LIN {X 0,Y 298.192,Z 478.827,A -85,B 0,C 180,E1 -16627.38,E2 -16627.38} C_VEL
LIN {X 0,Y 298.477,Z 490.19,A -85,B 0,C 180,E1 -16628.776,E2 -16628.776} C_VEL
LIN {X 0,Y 297.905,Z 495.3,A -85,B 0,C 180,E1 -16629.456,E2 -16629.456} C_VEL
LIN {X 0,Y 296.112,Z 505.168,A -85,B 0,C 180,E1 -16630.953,E2 -16630.953} C_VEL
LIN {X 0,Y 294.392,Z 514.617,A -85,B 0,C 180,E1 -16632.731,E2 -16632.731} C_VEL
LIN {X 0,Y 292.913,Z 523.059,A -85,B 0,C 180,E1 -16634.697,E2 -16634.697} C_VEL
LIN {X 0,Y 291.619,Z 530.199,A -85,B 0,C 180,E1 -16636.765,E2 -16636.765} C_VEL
LIN {X 0,Y 290.674,Z 535.95,A -85,B 0,C 180,E1 -16638.847,E2 -16638.847} C_VEL
LIN {X 0,Y 290.055,Z 540.511,A -85,B 0,C 180,E1 -16640.938,E2 -16640.938} C_VEL
LIN {X 0,Y 289.711,Z 543.998,A -85,B 0,C 180,E1 -16643.033,E2 -16643.033} C_VEL
LIN {X 0,Y 289.605,Z 545.749,A -85,B 0,C 180,E1 -16644.429,E2 -16644.429} C_VEL
LIN {X 0,Y 289.581,Z 547.097,A -85,B 0,C 180,E1 -16645.824,E2 -16645.824} C_VEL
LIN {X 0,Y 289.556,Z 548.044,A -85,B 0,C 180,E1 -16647.217,E2 -16647.217} C_VEL
LIN {X 0,Y 289.58,Z 548.554,A -85,B 0,C 180,E1 -16648.609,E2 -16648.609} C_VEL
LIN {X 0,Y 289.708,Z 548.659,A -85,B 0,C 180,E1 -16650,E2 -16650} C_VEL
LIN {X 0,Y 289.61,Z 548.356,A -85,B 0,C 180,E1 -16651.39,E2 -16651.39} C_VEL
LIN {X 0,Y 289.566,Z 547.661,A -85,B 0,C 180,E1 -16652.782,E2 -16652.782} C_VEL
LIN {X 0,Y 289.603,Z 546.528,A -85,B 0,C 180,E1 -16654.175,E2 -16654.175} C_VEL
LIN {X 0,Y 289.638,Z 544.641,A -85,B 0,C 180,E1 -16655.813,E2 -16655.813} C_VEL
LIN {X 0,Y 289.906,Z 540.509,A -85,B 0,C 180,E1 -16658.363,E2 -16658.363} C_VEL
LIN {X 0,Y 290.445,Z 535.873,A -85,B 0,C 180,E1 -16660.455,E2 -16660.455} C_VEL
LIN {X 0,Y 291.359,Z 528.848,A -85,B 0,C 180,E1 -16662.892,E2 -16662.892} C_VEL
LIN {X 0,Y 292.574,Z 521.257,A -85,B 0,C 180,E1 -16664.964,E2 -16664.964} C_VEL
LIN {X 0,Y 294.049,Z 512.473,A -85,B 0,C 180,E1 -16666.878,E2 -16666.878} C_VEL
LIN {X 0,Y 295.452,Z 501.889,A -85,B 0,C 180,E1 -16668.73,E2 -16668.73} C_VEL
LIN {X 0,Y 297.226,Z 490.969,A -85,B 0,C 180,E1 -16670.231,E2 -16670.231} C_VEL
LIN {X 0,Y 296.981,Z 482.707,A -85,B 0,C 180,E1 -16671.232,E2 -16671.232} C_VEL
LIN {X 0,Y 296.01,Z 470.906,A -85,B 0,C 180,E1 -16672.452,E2 -16672.452} C_VEL
LIN {X 0,Y 294.301,Z 457.671,A -85,B 0,C 180,E1 -16673.542,E2 -16673.542} C_VEL
LIN {X 0,Y 291.805,Z 444.082,A -85,B 0,C 180,E1 -16674.412,E2 -16674.412} C_VEL
LIN {X 0,Y 291.28,Z 441.289,A -85,B 0,C 180,E1 -16674.556,E2 -16674.556} C_VEL
LIN {X 0,Y 291.996,Z 435.686,A -85,B 0,C 180,E1 -16677.991,E2 -16677.991} C_VEL
LIN {X 0,Y 292.755,Z 430.711,A -85,B 0,C 180,E1 -16681.072,E2 -16681.072} C_VEL
LIN {X 0,Y 293.852,Z 424.513,A -85,B 0,C 180,E1 -16685.029,E2 -16685.029} C_VEL
LIN {X 0,Y 294.193,Z 422.009,A -85,B 0,C 180,E1 -16686.67,E2 -16686.67} C_VEL
LIN {X 0,Y 293.916,Z 418.336,A -85,B 0,C 180,E1 -16689.213,E2 -16689.213} C_VEL
LIN {X 0,Y 293.01,Z 413.146,A -85,B 0,C 180,E1 -16693.054,E2 -16693.054} C_VEL
LIN {X 0,Y 292.263,Z 409.186,A -85,B 0,C 180,E1 -16696.169,E2 -16696.169} C_VEL
LIN {X 0,Y 291.395,Z 404.188,A -85,B 0,C 180,E1 -16700.418,E2 -16700.418} C_VEL
LIN {X 0,Y 291.423,Z 404.186,A -85,B 0,C 180,E1 -16702.922,E2 -16702.922} C_VEL
LIN {X 0,Y 291.339,Z 404.193,A -85,B 0,C 180,E1 -16706.301,E2 -16706.301} C_VEL
LIN {X 0,Y 291.378,Z 404.189,A -85,B 0,C 180,E1 -16710.261,E2 -16710.261} C_VEL
LIN {X 0,Y 291.406,Z 404.185,A -85,B 0,C 180,E1 -16714.271,E2 -16714.271} C_VEL
LIN {X 0,Y 291.375,Z 404.189,A -85,B 0,C 180,E1 -16717.299,E2 -16717.299} C_VEL
LIN {X 0,Y 291.452,Z 404.179,A -85,B 0,C 180,E1 -16720.27,E2 -16720.27} C_VEL
LIN {X 0,Y 291.549,Z 404.17,A -85,B 0,C 180,E1 -16724.623,E2 -16724.623} C_VEL
LIN {X 0,Y 291.528,Z 404.172,A -85,B 0,C 180,E1 -16728.88,E2 -16728.88} C_VEL
LIN {X 0,Y 291.68,Z 404.149,A -85,B 0,C 180,E1 -16731.688,E2 -16731.688} C_VEL
LIN {X 0,Y 291.62,Z 404.158,A -85,B 0,C 180,E1 -16734.468,E2 -16734.468} C_VEL
LIN {X 0,Y 291.884,Z 404.129,A -85,B 0,C 180,E1 -16738.62,E2 -16738.62} C_VEL
LIN {X 0,Y 291.884,Z 404.123,A -85,B 0,C 180,E1 -16741.38,E2 -16741.38} C_VEL
LIN {X 0,Y 291.739,Z 404.144,A -85,B 0,C 180,E1 -16746.918,E2 -16746.918} C_VEL
LIN {X 0,Y 291.623,Z 404.156,A -85,B 0,C 180,E1 -16749.712,E2 -16749.712} C_VEL
LIN {X 0,Y 291.515,Z 404.167,A -85,B 0,C 180,E1 -16753.951,E2 -16753.951} C_VEL
LIN {X 0,Y 291.48,Z 404.176,A -85,B 0,C 180,E1 -16756.818,E2 -16756.818} C_VEL
LIN {X 0,Y 291.445,Z 404.179,A -85,B 0,C 180,E1 -16759.876,E2 -16759.876} C_VEL
LIN {X 0,Y 291.395,Z 404.185,A -85,B 0,C 180,E1 -16764.206,E2 -16764.206} C_VEL
LIN {X 0,Y 291.417,Z 404.182,A -85,B 0,C 180,E1 -16767.272,E2 -16767.272} C_VEL
LIN {X 0,Y 291.332,Z 404.194,A -85,B 0,C 180,E1 -16770.438,E2 -16770.438} C_VEL
LIN {X 0,Y 291.34,Z 404.19,A -85,B 0,C 180,E1 -16773.699,E2 -16773.699} C_VEL
LIN {X 0,Y 291.397,Z 404.185,A -85,B 0,C 180,E1 -16777.261,E2 -16777.261} C_VEL
LIN {X 0,Y 291.373,Z 404.186,A -85,B 0,C 180,E1 -16780.636,E2 -16780.636} C_VEL
LIN {X 0,Y 291.296,Z 404.201,A -85,B 0,C 180,E1 -16784.401,E2 -16784.401} C_VEL
LIN {X 0,Y 291.324,Z 404.194,A -85,B 0,C 180,E1 -16788.405,E2 -16788.405} C_VEL
LIN {X 0,Y 291.346,Z 404.184,A -85,B 0,C 180,E1 -16791.159,E2 -16791.159} C_VEL
LIN {X 0,Y 291.36,Z 404.188,A -85,B 0,C 180,E1 -16794.627,E2 -16794.627} C_VEL
LIN {X 0,Y 291.371,Z 404.193,A -85,B 0,C 180,E1 -16797.952,E2 -16797.952} C_VEL
LIN {X 0,Y 291.377,Z 404.187,A -85,B 0,C 180,E1 -16801.159,E2 -16801.159} C_VEL
LIN {X 0,Y 291.417,Z 404.18,A -85,B 0,C 180,E1 -16804.273,E2 -16804.273} C_VEL
LIN {X 0,Y 291.383,Z 404.186,A -85,B 0,C 180,E1 -16807.301,E2 -16807.301} C_VEL
LIN {X 0,Y 291.46,Z 404.178,A -85,B 0,C 180,E1 -16810.271,E2 -16810.271} C_VEL
LIN {X 0,Y 291.557,Z 404.165,A -85,B 0,C 180,E1 -16814.624,E2 -16814.624} C_VEL
LIN {X 0,Y 291.54,Z 404.165,A -85,B 0,C 180,E1 -16818.881,E2 -16818.881} C_VEL
LIN {X 0,Y 291.713,Z 404.15,A -85,B 0,C 180,E1 -16821.689,E2 -16821.689} C_VEL
LIN {X 0,Y 291.617,Z 404.157,A -85,B 0,C 180,E1 -16824.469,E2 -16824.469} C_VEL
LIN {X 0,Y 291.827,Z 404.132,A -85,B 0,C 180,E1 -16828.62,E2 -16828.62} C_VEL
LIN {X 0,Y 290.81,Z 404.574,A -85,B 0,C 180,E1 -16831.385,E2 -16831.385} C_VEL
LIN {X 0,Y 290.925,Z 406.775,A -85,B 0,C 180,E1 -16834.156,E2 -16834.156} C_VEL
LIN {X 0,Y 290.743,Z 409.661,A -85,B 0,C 180,E1 -16837.718,E2 -16837.718} C_VEL
LIN {X 0,Y 294.779,Z 423.834,A -85,B 0,C 180,E1 -16838.772,E2 -16838.772} C_VEL
LIN {X 0,Y 297.668,Z 435.363,A -85,B 0,C 180,E1 -16839.841,E2 -16839.841} C_VEL
LIN {X 0,Y 299.398,Z 444.412,A -85,B 0,C 180,E1 -16840.824,E2 -16840.824} C_VEL
LIN {X 0,Y 298.317,Z 455.723,A -85,B 0,C 180,E1 -16842.069,E2 -16842.069} C_VEL
LIN {X 0,Y 296.897,Z 466.255,A -85,B 0,C 180,E1 -16843.518,E2 -16843.518} C_VEL
LIN {X 0,Y 295.437,Z 475.921,A -85,B 0,C 180,E1 -16845.169,E2 -16845.169} C_VEL
LIN {X 0,Y 293.98,Z 484.669,A -85,B 0,C 180,E1 -16847.008,E2 -16847.008} C_VEL
LIN {X 0,Y 292.804,Z 491.976,A -85,B 0,C 180,E1 -16848.907,E2 -16848.907} C_VEL
LIN {X 0,Y 291.692,Z 498.923,A -85,B 0,C 180,E1 -16851.187,E2 -16851.187} C_VEL
LIN {X 0,Y 290.88,Z 504.062,A -85,B 0,C 180,E1 -16853.346,E2 -16853.346} C_VEL
LIN {X 0,Y 290.305,Z 508.488,A -85,B 0,C 180,E1 -16855.834,E2 -16855.834} C_VEL
LIN {X 0,Y 289.944,Z 510.535,A -85,B 0,C 180,E1 -16857.422,E2 -16857.422} C_VEL
LIN {X 0,Y 289.668,Z 512.157,A -85,B 0,C 180,E1 -16859.138,E2 -16859.138} C_VEL
LIN {X 0,Y 289.52,Z 513.41,A -85,B 0,C 180,E1 -16861.83,E2 -16861.83} C_VEL
LIN {X 0,Y 289.676,Z 513.225,A -85,B 0,C 180,E1 -16864.422,E2 -16864.422} C_VEL
LIN {X 0,Y 290.085,Z 511.76,A -85,B 0,C 180,E1 -16866.917,E2 -16866.917} C_VEL
LIN {X 0,Y 290.713,Z 509.081,A -85,B 0,C 180,E1 -16869.321,E2 -16869.321} C_VEL
LIN {X 0,Y 291.454,Z 505.271,A -85,B 0,C 180,E1 -16871.623,E2 -16871.623} C_VEL
LIN {X 0,Y 292.66,Z 499.549,A -85,B 0,C 180,E1 -16874.139,E2 -16874.139} C_VEL
LIN {X 0,Y 294.138,Z 492.812,A -85,B 0,C 180,E1 -16876.383,E2 -16876.383} C_VEL
LIN {X 0,Y 295.697,Z 485.104,A -85,B 0,C 180,E1 -16878.402,E2 -16878.402} C_VEL
LIN {X 0,Y 297.506,Z 475.704,A -85,B 0,C 180,E1 -16880.37,E2 -16880.37} C_VEL
LIN {X 0,Y 299.342,Z 465.228,A -85,B 0,C 180,E1 -16882.099,E2 -16882.099} C_VEL
LIN {X 0,Y 300.836,Z 455.272,A -85,B 0,C 180,E1 -16883.422,E2 -16883.422} C_VEL
LIN {X 0,Y 301.696,Z 448.206,A -85,B 0,C 180,E1 -16884.216,E2 -16884.216} C_VEL
LIN {X 0,Y 299.573,Z 437.974,A -85,B 0,C 180,E1 -16885.479,E2 -16885.479} C_VEL
LIN {X 0,Y 296.301,Z 426.472,A -85,B 0,C 180,E1 -16886.735,E2 -16886.735} C_VEL
LIN {X 0,Y 291.875,Z 414.797,A -85,B 0,C 180,E1 -16887.902,E2 -16887.902} C_VEL
LIN {X 0,Y 290.942,Z 412.026,A -85,B 0,C 180,E1 -16888.152,E2 -16888.152} C_VEL
LIN {X 0,Y 291.119,Z 409.938,A -85,B 0,C 180,E1 -16891.13,E2 -16891.13} C_VEL
LIN {X 0,Y 291.343,Z 407.807,A -85,B 0,C 180,E1 -16894.265,E2 -16894.265} C_VEL
LIN {X 0,Y 291.463,Z 405.839,A -85,B 0,C 180,E1 -16897.306,E2 -16897.306} C_VEL
LIN {X 0,Y 291.455,Z 404.184,A -85,B 0,C 180,E1 -16900.27,E2 -16900.27} C_VEL
LIN {X 0,Y 291.538,Z 404.173,A -85,B 0,C 180,E1 -16904.634,E2 -16904.634} C_VEL
LIN {X 0,Y 291.532,Z 404.17,A -85,B 0,C 180,E1 -16908.88,E2 -16908.88} C_VEL
LIN {X 0,Y 291.682,Z 404.153,A -85,B 0,C 180,E1 -16911.815,E2 -16911.815} C_VEL
LIN {X 0,Y 291.623,Z 404.157,A -85,B 0,C 180,E1 -16914.468,E2 -16914.468} C_VEL
LIN {X 0,Y 291.806,Z 404.133,A -85,B 0,C 180,E1 -16917.797,E2 -16917.797} C_VEL
LIN {X 0,Y 291.193,Z 404.214,A -85,B 0,C 180,E1 -16918.951,E2 -16918.951} C_VEL
LIN {X 0,Y 288.337,Z 404.57,A -85,B 0,C 180,E1 -16920.827,E2 -16920.827} C_VEL
LIN {X 0,Y 285.826,Z 404.878,A -85,B 0,C 180,E1 -16922.35,E2 -16922.35} C_VEL
LIN {X 0,Y 284.673,Z 405.026,A -85,B 0,C 180,E1 -16923.531,E2 -16923.531} C_VEL
LIN {X 0,Y 284.541,Z 405.039,A -85,B 0,C 180,E1 -16923.932,E2 -16923.932} C_VEL
LIN {X 0,Y 284.683,Z 405.023,A -85,B 0,C 180,E1 -16927.09,E2 -16927.09} C_VEL
LIN {X 0,Y 284.516,Z 405.043,A -85,B 0,C 180,E1 -16929.957,E2 -16929.957} C_VEL
LIN {X 0,Y 284.474,Z 405.049,A -85,B 0,C 180,E1 -16934.303,E2 -16934.303} C_VEL
LIN {X 0,Y 284.422,Z 405.056,A -85,B 0,C 180,E1 -16937.248,E2 -16937.248} C_VEL
LIN {X 0,Y 284.376,Z 405.063,A -85,B 0,C 180,E1 -16940.242,E2 -16940.242} C_VEL
LIN {X 0,Y 284.366,Z 405.065,A -85,B 0,C 180,E1 -16943.875,E2 -16943.875} C_VEL
LIN {X 0,Y 284.391,Z 405.059,A -85,B 0,C 180,E1 -16947.173,E2 -16947.173} C_VEL
LIN {X 0,Y 284.291,Z 405.073,A -85,B 0,C 180,E1 -16951.275,E2 -16951.275} C_VEL
LIN {X 0,Y 284.328,Z 405.111,A -85,B 0,C 180,E1 -16954.647,E2 -16954.647} C_VEL
LIN {X 0,Y 284.864,Z 407.869,A -85,B 0,C 180,E1 -16958.082,E2 -16958.082} C_VEL
LIN {X 0,Y 285.385,Z 411.197,A -85,B 0,C 180,E1 -16961.676,E2 -16961.676} C_VEL
LIN {X 0,Y 286.093,Z 415.045,A -85,B 0,C 180,E1 -16965.43,E2 -16965.43} C_VEL
LIN {X 0,Y 286.915,Z 419.566,A -85,B 0,C 180,E1 -16969.407,E2 -16969.407} C_VEL
LIN {X 0,Y 287.353,Z 423.183,A -85,B 0,C 180,E1 -16972.307,E2 -16972.307} C_VEL
LIN {X 0,Y 286.992,Z 426.701,A -85,B 0,C 180,E1 -16974.867,E2 -16974.867} C_VEL
LIN {X 0,Y 285.711,Z 433.39,A -85,B 0,C 180,E1 -16979.422,E2 -16979.422} C_VEL
LIN {X 0,Y 284.749,Z 439.073,A -85,B 0,C 180,E1 -16983.131,E2 -16983.131} C_VEL
LIN {X 0,Y 288.298,Z 453.543,A -85,B 0,C 180,E1 -16984.266,E2 -16984.266} C_VEL
LIN {X 0,Y 290.471,Z 465.856,A -85,B 0,C 180,E1 -16985.414,E2 -16985.414} C_VEL
LIN {X 0,Y 291.465,Z 477.28,A -85,B 0,C 180,E1 -16986.627,E2 -16986.627} C_VEL
LIN {X 0,Y 291.721,Z 488.901,A -85,B 0,C 180,E1 -16988.074,E2 -16988.074} C_VEL
LIN {X 0,Y 291.496,Z 494.105,A -85,B 0,C 180,E1 -16988.798,E2 -16988.798} C_VEL
LIN {X 0,Y 289.389,Z 505.1,A -85,B 0,C 180,E1 -16990.493,E2 -16990.493} C_VEL
LIN {X 0,Y 287.468,Z 515.166,A -85,B 0,C 180,E1 -16992.453,E2 -16992.453} C_VEL
LIN {X 0,Y 286.029,Z 522.874,A -85,B 0,C 180,E1 -16994.319,E2 -16994.319} C_VEL
LIN {X 0,Y 284.693,Z 529.951,A -85,B 0,C 180,E1 -16996.437,E2 -16996.437} C_VEL
LIN {X 0,Y 283.675,Z 535.656,A -85,B 0,C 180,E1 -16998.568,E2 -16998.568} C_VEL
LIN {X 0,Y 282.999,Z 540.176,A -85,B 0,C 180,E1 -17000.71,E2 -17000.71} C_VEL
LIN {X 0,Y 282.63,Z 543.631,A -85,B 0,C 180,E1 -17002.858,E2 -17002.858} C_VEL
LIN {X 0,Y 282.543,Z 545.371,A -85,B 0,C 180,E1 -17004.29,E2 -17004.29} C_VEL
LIN {X 0,Y 282.5,Z 546.707,A -85,B 0,C 180,E1 -17005.72,E2 -17005.72} C_VEL
LIN {X 0,Y 282.483,Z 547.638,A -85,B 0,C 180,E1 -17007.148,E2 -17007.148} C_VEL
LIN {X 0,Y 282.619,Z 548.22,A -85,B 0,C 180,E1 -17010,E2 -17010} C_VEL
LIN {X 0,Y 282.522,Z 547.905,A -85,B 0,C 180,E1 -17011.425,E2 -17011.425} C_VEL
LIN {X 0,Y 282.493,Z 547.195,A -85,B 0,C 180,E1 -17012.852,E2 -17012.852} C_VEL
LIN {X 0,Y 282.521,Z 546.036,A -85,B 0,C 180,E1 -17014.279,E2 -17014.279} C_VEL
LIN {X 0,Y 282.558,Z 544.359,A -85,B 0,C 180,E1 -17015.782,E2 -17015.782} C_VEL
LIN {X 0,Y 282.739,Z 541.243,A -85,B 0,C 180,E1 -17017.857,E2 -17017.857} C_VEL
LIN {X 0,Y 283.214,Z 536.959,A -85,B 0,C 180,E1 -17020.003,E2 -17020.003} C_VEL
LIN {X 0,Y 284.043,Z 530.454,A -85,B 0,C 180,E1 -17022.503,E2 -17022.503} C_VEL
LIN {X 0,Y 285.283,Z 523.33,A -85,B 0,C 180,E1 -17024.625,E2 -17024.625} C_VEL
LIN {X 0,Y 286.742,Z 514.44,A -85,B 0,C 180,E1 -17026.737,E2 -17026.737} C_VEL
LIN {X 0,Y 288.055,Z 505.319,A -85,B 0,C 180,E1 -17028.491,E2 -17028.491} C_VEL
LIN {X 0,Y 289.673,Z 495.289,A -85,B 0,C 180,E1 -17030.041,E2 -17030.041} C_VEL
LIN {X 0,Y 290.456,Z 490.049,A -85,B 0,C 180,E1 -17030.724,E2 -17030.724} C_VEL
LIN {X 0,Y 289.724,Z 477.737,A -85,B 0,C 180,E1 -17032.208,E2 -17032.208} C_VEL
LIN {X 0,Y 288.577,Z 465.951,A -85,B 0,C 180,E1 -17033.36,E2 -17033.36} C_VEL
LIN {X 0,Y 286.64,Z 453.247,A -85,B 0,C 180,E1 -17034.36,E2 -17034.36} C_VEL
LIN {X 0,Y 284.317,Z 440.877,A -85,B 0,C 180,E1 -17035.141,E2 -17035.141} C_VEL
LIN {X 0,Y 285.104,Z 435.166,A -85,B 0,C 180,E1 -17038.729,E2 -17038.729} C_VEL
LIN {X 0,Y 285.884,Z 430.222,A -85,B 0,C 180,E1 -17041.906,E2 -17041.906} C_VEL
LIN {X 0,Y 286.829,Z 425.249,A -85,B 0,C 180,E1 -17045.155,E2 -17045.155} C_VEL
LIN {X 0,Y 287.146,Z 421.493,A -85,B 0,C 180,E1 -17047.724,E2 -17047.724} C_VEL
LIN {X 0,Y 286.6,Z 417.651,A -85,B 0,C 180,E1 -17050.52,E2 -17050.52} C_VEL
LIN {X 0,Y 285.695,Z 412.534,A -85,B 0,C 180,E1 -17054.488,E2 -17054.488} C_VEL
LIN {X 0,Y 284.666,Z 406.967,A -85,B 0,C 180,E1 -17059.138,E2 -17059.138} C_VEL
LIN {X 0,Y 284.34,Z 405.068,A -85,B 0,C 180,E1 -17060.929,E2 -17060.929} C_VEL
LIN {X 0,Y 284.357,Z 405.066,A -85,B 0,C 180,E1 -17064.645,E2 -17064.645} C_VEL
LIN {X 0,Y 284.288,Z 405.075,A -85,B 0,C 180,E1 -17068.725,E2 -17068.725} C_VEL
LIN {X 0,Y 284.388,Z 405.064,A -85,B 0,C 180,E1 -17072.827,E2 -17072.827} C_VEL
LIN {X 0,Y 284.36,Z 405.065,A -85,B 0,C 180,E1 -17076.706,E2 -17076.706} C_VEL
LIN {X 0,Y 284.397,Z 405.058,A -85,B 0,C 180,E1 -17081.261,E2 -17081.261} C_VEL
LIN {X 0,Y 284.486,Z 405.048,A -85,B 0,C 180,E1 -17084.459,E2 -17084.459} C_VEL
LIN {X 0,Y 284.48,Z 405.05,A -85,B 0,C 180,E1 -17088.601,E2 -17088.601} C_VEL
LIN {X 0,Y 284.632,Z 405.027,A -85,B 0,C 180,E1 -17091.48,E2 -17091.48} C_VEL
LIN {X 0,Y 284.591,Z 405.032,A -85,B 0,C 180,E1 -17094.331,E2 -17094.331} C_VEL
LIN {X 0,Y 284.85,Z 405.005,A -85,B 0,C 180,E1 -17098.586,E2 -17098.586} C_VEL
LIN {X 0,Y 284.85,Z 404.998,A -85,B 0,C 180,E1 -17101.414,E2 -17101.414} C_VEL
LIN {X 0,Y 284.691,Z 405.021,A -85,B 0,C 180,E1 -17107.09,E2 -17107.09} C_VEL
LIN {X 0,Y 284.56,Z 405.037,A -85,B 0,C 180,E1 -17109.956,E2 -17109.956} C_VEL
LIN {X 0,Y 284.471,Z 405.047,A -85,B 0,C 180,E1 -17114.304,E2 -17114.304} C_VEL
LIN {X 0,Y 284.419,Z 405.054,A -85,B 0,C 180,E1 -17117.249,E2 -17117.249} C_VEL
LIN {X 0,Y 284.373,Z 405.063,A -85,B 0,C 180,E1 -17120.243,E2 -17120.243} C_VEL
LIN {X 0,Y 284.363,Z 405.058,A -85,B 0,C 180,E1 -17123.876,E2 -17123.876} C_VEL
LIN {X 0,Y 284.392,Z 405.057,A -85,B 0,C 180,E1 -17127.174,E2 -17127.174} C_VEL
LIN {X 0,Y 284.291,Z 405.067,A -85,B 0,C 180,E1 -17131.275,E2 -17131.275} C_VEL
LIN {X 0,Y 284.358,Z 405.061,A -85,B 0,C 180,E1 -17135.355,E2 -17135.355} C_VEL
LIN {X 0,Y 284.329,Z 405.07,A -85,B 0,C 180,E1 -17138.167,E2 -17138.167} C_VEL
LIN {X 0,Y 284.289,Z 405.069,A -85,B 0,C 180,E1 -17141.873,E2 -17141.873} C_VEL
LIN {X 0,Y 284.253,Z 405.079,A -85,B 0,C 180,E1 -17146.19,E2 -17146.19} C_VEL
LIN {X 0,Y 284.304,Z 405.066,A -85,B 0,C 180,E1 -17150.025,E2 -17150.025} C_VEL
LIN {X 0,Y 284.329,Z 405.058,A -85,B 0,C 180,E1 -17153.615,E2 -17153.615} C_VEL
LIN {X 0,Y 284.307,Z 405.068,A -85,B 0,C 180,E1 -17157.191,E2 -17157.191} C_VEL
LIN {X 0,Y 284.355,Z 405.064,A -85,B 0,C 180,E1 -17160.377,E2 -17160.377} C_VEL
LIN {X 0,Y 284.378,Z 405.057,A -85,B 0,C 180,E1 -17163.588,E2 -17163.588} C_VEL
LIN {X 0,Y 284.368,Z 405.059,A -85,B 0,C 180,E1 -17166.708,E2 -17166.708} C_VEL
LIN {X 0,Y 284.405,Z 405.055,A -85,B 0,C 180,E1 -17171.263,E2 -17171.263} C_VEL
LIN {X 0,Y 284.494,Z 405.045,A -85,B 0,C 180,E1 -17174.46,E2 -17174.46} C_VEL
LIN {X 0,Y 284.491,Z 405.043,A -85,B 0,C 180,E1 -17178.602,E2 -17178.602} C_VEL
LIN {X 0,Y 284.663,Z 405.027,A -85,B 0,C 180,E1 -17181.482,E2 -17181.482} C_VEL
LIN {X 0,Y 284.59,Z 405.033,A -85,B 0,C 180,E1 -17184.332,E2 -17184.332} C_VEL
LIN {X 0,Y 284.789,Z 405.008,A -85,B 0,C 180,E1 -17188.586,E2 -17188.586} C_VEL
LIN {X 0,Y 283.768,Z 405.542,A -85,B 0,C 180,E1 -17191.42,E2 -17191.42} C_VEL
LIN {X 0,Y 283.887,Z 407.745,A -85,B 0,C 180,E1 -17194.259,E2 -17194.259} C_VEL
LIN {X 0,Y 283.716,Z 410.111,A -85,B 0,C 180,E1 -17197.161,E2 -17197.161} C_VEL
LIN {X 0,Y 287.713,Z 423.844,A -85,B 0,C 180,E1 -17198.217,E2 -17198.217} C_VEL
LIN {X 0,Y 290.911,Z 436.611,A -85,B 0,C 180,E1 -17199.439,E2 -17199.439} C_VEL
LIN {X 0,Y 292.666,Z 446.475,A -85,B 0,C 180,E1 -17200.551,E2 -17200.551} C_VEL
LIN {X 0,Y 291.37,Z 457.536,A -85,B 0,C 180,E1 -17201.831,E2 -17201.831} C_VEL
LIN {X 0,Y 289.792,Z 468.719,A -85,B 0,C 180,E1 -17203.462,E2 -17203.462} C_VEL
LIN {X 0,Y 288.273,Z 478.258,A -85,B 0,C 180,E1 -17205.194,E2 -17205.194} C_VEL
LIN {X 0,Y 286.801,Z 486.78,A -85,B 0,C 180,E1 -17207.119,E2 -17207.119} C_VEL
LIN {X 0,Y 285.431,Z 494.876,A -85,B 0,C 180,E1 -17209.415,E2 -17209.415} C_VEL
LIN {X 0,Y 284.35,Z 501.337,A -85,B 0,C 180,E1 -17211.761,E2 -17211.761} C_VEL
LIN {X 0,Y 283.56,Z 506.404,A -85,B 0,C 180,E1 -17214.191,E2 -17214.191} C_VEL
LIN {X 0,Y 283.032,Z 510.101,A -85,B 0,C 180,E1 -17216.629,E2 -17216.629} C_VEL
LIN {X 0,Y 282.706,Z 511.814,A -85,B 0,C 180,E1 -17218.186,E2 -17218.186} C_VEL
LIN {X 0,Y 282.518,Z 513.04,A -85,B 0,C 180,E1 -17219.836,E2 -17219.836} C_VEL
LIN {X 0,Y 282.432,Z 513.897,A -85,B 0,C 180,E1 -17222.214,E2 -17222.214} C_VEL
LIN {X 0,Y 282.656,Z 513.566,A -85,B 0,C 180,E1 -17224.881,E2 -17224.881} C_VEL
LIN {X 0,Y 283.124,Z 511.934,A -85,B 0,C 180,E1 -17227.407,E2 -17227.407} C_VEL
LIN {X 0,Y 283.882,Z 508.804,A -85,B 0,C 180,E1 -17230.066,E2 -17230.066} C_VEL
LIN {X 0,Y 284.618,Z 505.178,A -85,B 0,C 180,E1 -17232.201,E2 -17232.201} C_VEL
LIN {X 0,Y 285.781,Z 499.981,A -85,B 0,C 180,E1 -17234.506,E2 -17234.506} C_VEL
LIN {X 0,Y 287.313,Z 493.347,A -85,B 0,C 180,E1 -17236.771,E2 -17236.771} C_VEL
LIN {X 0,Y 289.111,Z 485.063,A -85,B 0,C 180,E1 -17238.978,E2 -17238.978} C_VEL
LIN {X 0,Y 291.009,Z 475.574,A -85,B 0,C 180,E1 -17240.987,E2 -17240.987} C_VEL
LIN {X 0,Y 292.814,Z 465.777,A -85,B 0,C 180,E1 -17242.626,E2 -17242.626} C_VEL
LIN {X 0,Y 294.471,Z 455.215,A -85,B 0,C 180,E1 -17244.051,E2 -17244.051} C_VEL
LIN {X 0,Y 295.117,Z 449.319,A -85,B 0,C 180,E1 -17244.737,E2 -17244.737} C_VEL
LIN {X 0,Y 292.891,Z 438.87,A -85,B 0,C 180,E1 -17246.09,E2 -17246.09} C_VEL
LIN {X 0,Y 289.435,Z 426.934,A -85,B 0,C 180,E1 -17247.466,E2 -17247.466} C_VEL
LIN {X 0,Y 285.051,Z 415.59,A -85,B 0,C 180,E1 -17248.663,E2 -17248.663} C_VEL
LIN {X 0,Y 283.974,Z 412.528,A -85,B 0,C 180,E1 -17248.959,E2 -17248.959} C_VEL
LIN {X 0,Y 284.248,Z 409.868,A -85,B 0,C 180,E1 -17252.884,E2 -17252.884} C_VEL
LIN {X 0,Y 284.444,Z 407.426,A -85,B 0,C 180,E1 -17256.713,E2 -17256.713} C_VEL
LIN {X 0,Y 284.435,Z 405.546,A -85,B 0,C 180,E1 -17259.87,E2 -17259.87} C_VEL
LIN {X 0,Y 284.395,Z 405.062,A -85,B 0,C 180,E1 -17261.261,E2 -17261.261} C_VEL
LIN {X 0,Y 284.475,Z 405.052,A -85,B 0,C 180,E1 -17264.469,E2 -17264.469} C_VEL
LIN {X 0,Y 284.484,Z 405.048,A -85,B 0,C 180,E1 -17268.601,E2 -17268.601} C_VEL
LIN {X 0,Y 284.636,Z 405.031,A -85,B 0,C 180,E1 -17271.48,E2 -17271.48} C_VEL
LIN {X 0,Y 284.594,Z 405.033,A -85,B 0,C 180,E1 -17274.331,E2 -17274.331} C_VEL
LIN {X 0,Y 284.852,Z 405.004,A -85,B 0,C 180,E1 -17278.586,E2 -17278.586} C_VEL
LIN {X 0,Y 284.853,Z 405.003,A -85,B 0,C 180,E1 -17281.414,E2 -17281.414} C_VEL
LIN {X 0,Y 284.541,Z 405.039,A -85,B 0,C 180,E1 -17283.932,E2 -17283.932} C_VEL
LIN {X 0,Y 283.79,Z 405.139,A -85,B 0,C 180,E1 -17285.114,E2 -17285.114} C_VEL
LIN {X 0,Y 280.97,Z 405.494,A -85,B 0,C 180,E1 -17287.041,E2 -17287.041} C_VEL
LIN {X 0,Y 278.61,Z 405.784,A -85,B 0,C 180,E1 -17288.606,E2 -17288.606} C_VEL
LIN {X 0,Y 277.564,Z 405.909,A -85,B 0,C 180,E1 -17289.816,E2 -17289.816} C_VEL
LIN {X 0,Y 277.457,Z 405.92,A -85,B 0,C 180,E1 -17290.226,E2 -17290.226} C_VEL
LIN {X 0,Y 277.425,Z 405.928,A -85,B 0,C 180,E1 -17294.675,E2 -17294.675} C_VEL
LIN {X 0,Y 277.342,Z 405.934,A -85,B 0,C 180,E1 -17299.234,E2 -17299.234} C_VEL
LIN {X 0,Y 277.316,Z 405.943,A -85,B 0,C 180,E1 -17304.17,E2 -17304.17} C_VEL
LIN {X 0,Y 277.32,Z 405.942,A -85,B 0,C 180,E1 -17307.504,E2 -17307.504} C_VEL
LIN {X 0,Y 277.27,Z 405.948,A -85,B 0,C 180,E1 -17310.482,E2 -17310.482} C_VEL
LIN {X 0,Y 277.261,Z 405.952,A -85,B 0,C 180,E1 -17313.496,E2 -17313.496} C_VEL
LIN {X 0,Y 277.826,Z 408.899,A -85,B 0,C 180,E1 -17317.381,E2 -17317.381} C_VEL
LIN {X 0,Y 278.331,Z 412.111,A -85,B 0,C 180,E1 -17321.035,E2 -17321.035} C_VEL
LIN {X 0,Y 279.094,Z 416.179,A -85,B 0,C 180,E1 -17325.165,E2 -17325.165} C_VEL
LIN {X 0,Y 279.918,Z 420.681,A -85,B 0,C 180,E1 -17329.248,E2 -17329.248} C_VEL
LIN {X 0,Y 280.368,Z 424.167,A -85,B 0,C 180,E1 -17332.111,E2 -17332.111} C_VEL
LIN {X 0,Y 280.333,Z 425.75,A -85,B 0,C 180,E1 -17333.345,E2 -17333.345} C_VEL
LIN {X 0,Y 279.461,Z 430.007,A -85,B 0,C 180,E1 -17336.409,E2 -17336.409} C_VEL
LIN {X 0,Y 278.326,Z 435.931,A -85,B 0,C 180,E1 -17340.502,E2 -17340.502} C_VEL
LIN {X 0,Y 277.875,Z 438.585,A -85,B 0,C 180,E1 -17342.279,E2 -17342.279} C_VEL
LIN {X 0,Y 279.538,Z 444.902,A -85,B 0,C 180,E1 -17342.776,E2 -17342.776} C_VEL
LIN {X 0,Y 282.351,Z 456.878,A -85,B 0,C 180,E1 -17343.849,E2 -17343.849} C_VEL
LIN {X 0,Y 284.115,Z 468.137,A -85,B 0,C 180,E1 -17344.977,E2 -17344.977} C_VEL
LIN {X 0,Y 284.962,Z 480.077,A -85,B 0,C 180,E1 -17346.342,E2 -17346.342} C_VEL
LIN {X 0,Y 285.022,Z 491.674,A -85,B 0,C 180,E1 -17347.912,E2 -17347.912} C_VEL
LIN {X 0,Y 284.429,Z 496.544,A -85,B 0,C 180,E1 -17348.626,E2 -17348.626} C_VEL
LIN {X 0,Y 282.303,Z 507.009,A -85,B 0,C 180,E1 -17350.362,E2 -17350.362} C_VEL
LIN {X 0,Y 280.558,Z 515.661,A -85,B 0,C 180,E1 -17352.158,E2 -17352.158} C_VEL
LIN {X 0,Y 278.912,Z 523.93,A -85,B 0,C 180,E1 -17354.283,E2 -17354.283} C_VEL
LIN {X 0,Y 277.538,Z 530.73,A -85,B 0,C 180,E1 -17356.453,E2 -17356.453} C_VEL
LIN {X 0,Y 276.4,Z 537.015,A -85,B 0,C 180,E1 -17359.006,E2 -17359.006} C_VEL
LIN {X 0,Y 275.815,Z 541.135,A -85,B 0,C 180,E1 -17361.206,E2 -17361.206} C_VEL
LIN {X 0,Y 275.579,Z 543.28,A -85,B 0,C 180,E1 -17362.674,E2 -17362.674} C_VEL
LIN {X 0,Y 275.443,Z 545.193,A -85,B 0,C 180,E1 -17364.324,E2 -17364.324} C_VEL
LIN {X 0,Y 275.411,Z 547.232,A -85,B 0,C 180,E1 -17367.074,E2 -17367.074} C_VEL
LIN {X 0,Y 275.53,Z 547.78,A -85,B 0,C 180,E1 -17370,E2 -17370} C_VEL
LIN {X 0,Y 275.438,Z 547.452,A -85,B 0,C 180,E1 -17371.462,E2 -17371.462} C_VEL
LIN {X 0,Y 275.422,Z 546.724,A -85,B 0,C 180,E1 -17372.925,E2 -17372.925} C_VEL
LIN {X 0,Y 275.442,Z 545.541,A -85,B 0,C 180,E1 -17374.39,E2 -17374.39} C_VEL
LIN {X 0,Y 275.514,Z 542.987,A -85,B 0,C 180,E1 -17376.591,E2 -17376.591} C_VEL
LIN {X 0,Y 275.822,Z 539.402,A -85,B 0,C 180,E1 -17378.793,E2 -17378.793} C_VEL
LIN {X 0,Y 276.387,Z 534.691,A -85,B 0,C 180,E1 -17380.994,E2 -17380.994} C_VEL
LIN {X 0,Y 277.492,Z 527.595,A -85,B 0,C 180,E1 -17383.548,E2 -17383.548} C_VEL
LIN {X 0,Y 278.818,Z 519.901,A -85,B 0,C 180,E1 -17385.721,E2 -17385.721} C_VEL
LIN {X 0,Y 280.405,Z 510.407,A -85,B 0,C 180,E1 -17387.842,E2 -17387.842} C_VEL
LIN {X 0,Y 281.817,Z 501.326,A -85,B 0,C 180,E1 -17389.484,E2 -17389.484} C_VEL
LIN {X 0,Y 283.536,Z 490.465,A -85,B 0,C 180,E1 -17391.063,E2 -17391.063} C_VEL
LIN {X 0,Y 282.852,Z 478.198,A -85,B 0,C 180,E1 -17392.598,E2 -17392.598} C_VEL
LIN {X 0,Y 281.632,Z 465.578,A -85,B 0,C 180,E1 -17393.881,E2 -17393.881} C_VEL
LIN {X 0,Y 279.705,Z 452.813,A -85,B 0,C 180,E1 -17394.918,E2 -17394.918} C_VEL
LIN {X 0,Y 277.353,Z 440.473,A -85,B 0,C 180,E1 -17395.717,E2 -17395.717} C_VEL
LIN {X 0,Y 278.444,Z 433.413,A -85,B 0,C 180,E1 -17400.317,E2 -17400.317} C_VEL
LIN {X 0,Y 279.596,Z 427.119,A -85,B 0,C 180,E1 -17404.518,E2 -17404.518} C_VEL
LIN {X 0,Y 280.129,Z 423.493,A -85,B 0,C 180,E1 -17407.021,E2 -17407.021} C_VEL
LIN {X 0,Y 279.742,Z 419.663,A -85,B 0,C 180,E1 -17409.837,E2 -17409.837} C_VEL
LIN {X 0,Y 278.792,Z 414.276,A -85,B 0,C 180,E1 -17414.074,E2 -17414.074} C_VEL
LIN {X 0,Y 278.092,Z 410.627,A -85,B 0,C 180,E1 -17417.128,E2 -17417.128} C_VEL
LIN {X 0,Y 277.289,Z 405.945,A -85,B 0,C 180,E1 -17421.297,E2 -17421.297} C_VEL
LIN {X 0,Y 277.299,Z 405.944,A -85,B 0,C 180,E1 -17424.344,E2 -17424.344} C_VEL
LIN {X 0,Y 277.238,Z 405.95,A -85,B 0,C 180,E1 -17427.836,E2 -17427.836} C_VEL
LIN {X 0,Y 277.28,Z 405.947,A -85,B 0,C 180,E1 -17431.212,E2 -17431.212} C_VEL
LIN {X 0,Y 277.305,Z 405.943,A -85,B 0,C 180,E1 -17434.479,E2 -17434.479} C_VEL
LIN {X 0,Y 277.279,Z 405.944,A -85,B 0,C 180,E1 -17437.654,E2 -17437.654} C_VEL
LIN {X 0,Y 277.339,Z 405.941,A -85,B 0,C 180,E1 -17440.766,E2 -17440.766} C_VEL
LIN {X 0,Y 277.428,Z 405.926,A -85,B 0,C 180,E1 -17445.326,E2 -17445.326} C_VEL
LIN {X 0,Y 277.454,Z 405.922,A -85,B 0,C 180,E1 -17449.787,E2 -17449.787} C_VEL
LIN {X 0,Y 277.634,Z 405.901,A -85,B 0,C 180,E1 -17452.729,E2 -17452.729} C_VEL
LIN {X 0,Y 277.816,Z 405.881,A -85,B 0,C 180,E1 -17458.551,E2 -17458.551} C_VEL
LIN {X 0,Y 277.816,Z 405.874,A -85,B 0,C 180,E1 -17461.45,E2 -17461.45} C_VEL
LIN {X 0,Y 277.646,Z 405.898,A -85,B 0,C 180,E1 -17467.271,E2 -17467.271} C_VEL
LIN {X 0,Y 277.5,Z 405.918,A -85,B 0,C 180,E1 -17470.212,E2 -17470.212} C_VEL
LIN {X 0,Y 277.422,Z 405.927,A -85,B 0,C 180,E1 -17474.675,E2 -17474.675} C_VEL
LIN {X 0,Y 277.339,Z 405.936,A -85,B 0,C 180,E1 -17479.234,E2 -17479.234} C_VEL
LIN {X 0,Y 277.314,Z 405.938,A -85,B 0,C 180,E1 -17484.171,E2 -17484.171} C_VEL
LIN {X 0,Y 277.321,Z 405.938,A -85,B 0,C 180,E1 -17487.506,E2 -17487.506} C_VEL
LIN {X 0,Y 277.268,Z 405.945,A -85,B 0,C 180,E1 -17490.482,E2 -17490.482} C_VEL
LIN {X 0,Y 277.25,Z 405.945,A -85,B 0,C 180,E1 -17493.896,E2 -17493.896} C_VEL
LIN {X 0,Y 277.284,Z 405.943,A -85,B 0,C 180,E1 -17497.467,E2 -17497.467} C_VEL
LIN {X 0,Y 277.231,Z 405.945,A -85,B 0,C 180,E1 -17501.233,E2 -17501.233} C_VEL
LIN {X 0,Y 277.201,Z 405.953,A -85,B 0,C 180,E1 -17505.227,E2 -17505.227} C_VEL
LIN {X 0,Y 277.22,Z 405.948,A -85,B 0,C 180,E1 -17509.513,E2 -17509.513} C_VEL
LIN {X 0,Y 277.263,Z 405.937,A -85,B 0,C 180,E1 -17512.531,E2 -17512.531} C_VEL
LIN {X 0,Y 277.246,Z 405.95,A -85,B 0,C 180,E1 -17516.105,E2 -17516.105} C_VEL
LIN {X 0,Y 277.261,Z 405.949,A -85,B 0,C 180,E1 -17519.54,E2 -17519.54} C_VEL
LIN {X 0,Y 277.358,Z 405.93,A -85,B 0,C 180,E1 -17522.865,E2 -17522.865} C_VEL
LIN {X 0,Y 277.33,Z 405.937,A -85,B 0,C 180,E1 -17526.081,E2 -17526.081} C_VEL
LIN {X 0,Y 277.347,Z 405.934,A -85,B 0,C 180,E1 -17530.767,E2 -17530.767} C_VEL
LIN {X 0,Y 277.437,Z 405.925,A -85,B 0,C 180,E1 -17535.327,E2 -17535.327} C_VEL
LIN {X 0,Y 277.509,Z 405.916,A -85,B 0,C 180,E1 -17539.789,E2 -17539.789} C_VEL
LIN {X 0,Y 277.657,Z 405.897,A -85,B 0,C 180,E1 -17542.73,E2 -17542.73} C_VEL
LIN {X 0,Y 277.751,Z 405.885,A -85,B 0,C 180,E1 -17548.55,E2 -17548.55} C_VEL
LIN {X 0,Y 277.108,Z 405.969,A -85,B 0,C 180,E1 -17550,E2 -17550} C_VEL
LIN {X 0,Y 276.725,Z 406.51,A -85,B 0,C 180,E1 -17551.456,E2 -17551.456} C_VEL
LIN {X 0,Y 276.849,Z 408.714,A -85,B 0,C 180,E1 -17554.368,E2 -17554.368} C_VEL
LIN {X 0,Y 276.693,Z 410.467,A -85,B 0,C 180,E1 -17556.563,E2 -17556.563} C_VEL
LIN {X 0,Y 280.881,Z 424.737,A -85,B 0,C 180,E1 -17557.709,E2 -17557.709} C_VEL
LIN {X 0,Y 283.908,Z 436.733,A -85,B 0,C 180,E1 -17558.901,E2 -17558.901} C_VEL
LIN {X 0,Y 285.848,Z 447.114,A -85,B 0,C 180,E1 -17560.111,E2 -17560.111} C_VEL
LIN {X 0,Y 284.635,Z 457.869,A -85,B 0,C 180,E1 -17561.393,E2 -17561.393} C_VEL
LIN {X 0,Y 283.133,Z 468.15,A -85,B 0,C 180,E1 -17562.909,E2 -17562.909} C_VEL
LIN {X 0,Y 281.73,Z 476.685,A -85,B 0,C 180,E1 -17564.446,E2 -17564.446} C_VEL
LIN {X 0,Y 280.211,Z 485.393,A -85,B 0,C 180,E1 -17566.36,E2 -17566.36} C_VEL
LIN {X 0,Y 278.904,Z 492.768,A -85,B 0,C 180,E1 -17568.36,E2 -17568.36} C_VEL
LIN {X 0,Y 277.694,Z 499.736,A -85,B 0,C 180,E1 -17570.752,E2 -17570.752} C_VEL
LIN {X 0,Y 276.775,Z 505.04,A -85,B 0,C 180,E1 -17573.095,E2 -17573.095} C_VEL
LIN {X 0,Y 276.169,Z 509.331,A -85,B 0,C 180,E1 -17575.634,E2 -17575.634} C_VEL
LIN {X 0,Y 275.796,Z 511.385,A -85,B 0,C 180,E1 -17577.302,E2 -17577.302} C_VEL
LIN {X 0,Y 275.431,Z 513.461,A -85,B 0,C 180,E1 -17579.823,E2 -17579.823} C_VEL
LIN {X 0,Y 275.384,Z 514.386,A -85,B 0,C 180,E1 -17582.628,E2 -17582.628} C_VEL
LIN {X 0,Y 275.622,Z 513.874,A -85,B 0,C 180,E1 -17585.317,E2 -17585.317} C_VEL
LIN {X 0,Y 276.15,Z 512.094,A -85,B 0,C 180,E1 -17587.912,E2 -17587.912} C_VEL
LIN {X 0,Y 276.904,Z 509.151,A -85,B 0,C 180,E1 -17590.41,E2 -17590.41} C_VEL
LIN {X 0,Y 277.943,Z 504.614,A -85,B 0,C 180,E1 -17593.056,E2 -17593.056} C_VEL
LIN {X 0,Y 279.124,Z 499.736,A -85,B 0,C 180,E1 -17595.17,E2 -17595.17} C_VEL
LIN {X 0,Y 280.722,Z 492.935,A -85,B 0,C 180,E1 -17597.471,E2 -17597.471} C_VEL
LIN {X 0,Y 282.314,Z 485.979,A -85,B 0,C 180,E1 -17599.357,E2 -17599.357} C_VEL
LIN {X 0,Y 284.105,Z 477.683,A -85,B 0,C 180,E1 -17601.189,E2 -17601.189} C_VEL
LIN {X 0,Y 286.063,Z 467.624,A -85,B 0,C 180,E1 -17602.982,E2 -17602.982} C_VEL
LIN {X 0,Y 287.86,Z 456.936,A -85,B 0,C 180,E1 -17604.489,E2 -17604.489} C_VEL
LIN {X 0,Y 288.629,Z 451.859,A -85,B 0,C 180,E1 -17605.095,E2 -17605.095} C_VEL
LIN {X 0,Y 287.02,Z 443.031,A -85,B 0,C 180,E1 -17606.314,E2 -17606.314} C_VEL
LIN {X 0,Y 284.175,Z 432.227,A -85,B 0,C 180,E1 -17607.668,E2 -17607.668} C_VEL
LIN {X 0,Y 280.095,Z 420.767,A -85,B 0,C 180,E1 -17608.992,E2 -17608.992} C_VEL
LIN {X 0,Y 277.089,Z 413.521,A -85,B 0,C 180,E1 -17609.775,E2 -17609.775} C_VEL
LIN {X 0,Y 277.01,Z 413.031,A -85,B 0,C 180,E1 -17609.838,E2 -17609.838} C_VEL
LIN {X 0,Y 277.243,Z 411.054,A -85,B 0,C 180,E1 -17612.851,E2 -17612.851} C_VEL
LIN {X 0,Y 277.449,Z 409.015,A -85,B 0,C 180,E1 -17616.09,E2 -17616.09} C_VEL
LIN {X 0,Y 277.428,Z 406.976,A -85,B 0,C 180,E1 -17619.603,E2 -17619.603} C_VEL
LIN {X 0,Y 277.355,Z 405.938,A -85,B 0,C 180,E1 -17622.297,E2 -17622.297} C_VEL
LIN {X 0,Y 277.425,Z 405.929,A -85,B 0,C 180,E1 -17625.325,E2 -17625.325} C_VEL
LIN {X 0,Y 277.458,Z 405.925,A -85,B 0,C 180,E1 -17629.787,E2 -17629.787} C_VEL
LIN {X 0,Y 277.637,Z 405.899,A -85,B 0,C 180,E1 -17632.728,E2 -17632.728} C_VEL
LIN {X 0,Y 277.818,Z 405.88,A -85,B 0,C 180,E1 -17638.55,E2 -17638.55} C_VEL
LIN {X 0,Y 277.819,Z 405.879,A -85,B 0,C 180,E1 -17641.449,E2 -17641.449} C_VEL
LIN {X 0,Y 277.637,Z 405.899,A -85,B 0,C 180,E1 -17647.271,E2 -17647.271} C_VEL
LIN {X 0,Y 277.457,Z 405.92,A -85,B 0,C 180,E1 -17650.226,E2 -17650.226} C_VEL
LIN {X 0,Y 276.746,Z 406.012,A -85,B 0,C 180,E1 -17651.437,E2 -17651.437} C_VEL
LIN {X 0,Y 273.93,Z 406.361,A -85,B 0,C 180,E1 -17653.41,E2 -17653.41} C_VEL
LIN {X 0,Y 270.712,Z 406.763,A -85,B 0,C 180,E1 -17655.836,E2 -17655.836} C_VEL
LIN {X 0,Y 270.344,Z 406.805,A -85,B 0,C 180,E1 -17656.674,E2 -17656.674} C_VEL
LIN {X 0,Y 270.29,Z 406.817,A -85,B 0,C 180,E1 -17660.602,E2 -17660.602} C_VEL
LIN {X 0,Y 270.271,Z 406.82,A -85,B 0,C 180,E1 -17664.586,E2 -17664.586} C_VEL
LIN {X 0,Y 270.267,Z 406.821,A -85,B 0,C 180,E1 -17667.909,E2 -17667.909} C_VEL
LIN {X 0,Y 270.203,Z 406.921,A -85,B 0,C 180,E1 -17672.443,E2 -17672.443} C_VEL
LIN {X 0,Y 270.809,Z 409.948,A -85,B 0,C 180,E1 -17676.648,E2 -17676.648} C_VEL
LIN {X 0,Y 271.291,Z 413.06,A -85,B 0,C 180,E1 -17680.364,E2 -17680.364} C_VEL
LIN {X 0,Y 271.927,Z 416.71,A -85,B 0,C 180,E1 -17684.252,E2 -17684.252} C_VEL
LIN {X 0,Y 272.755,Z 421.004,A -85,B 0,C 180,E1 -17688.351,E2 -17688.351} C_VEL
LIN {X 0,Y 273.349,Z 425.111,A -85,B 0,C 180,E1 -17691.899,E2 -17691.899} C_VEL
LIN {X 0,Y 273.003,Z 428.596,A -85,B 0,C 180,E1 -17694.604,E2 -17694.604} C_VEL
LIN {X 0,Y 271.753,Z 434.481,A -85,B 0,C 180,E1 -17698.853,E2 -17698.853} C_VEL
LIN {X 0,Y 271.018,Z 438.082,A -85,B 0,C 180,E1 -17701.372,E2 -17701.372} C_VEL
LIN {X 0,Y 272.829,Z 444.759,A -85,B 0,C 180,E1 -17701.932,E2 -17701.932} C_VEL
LIN {X 0,Y 275.782,Z 457.313,A -85,B 0,C 180,E1 -17703.118,E2 -17703.118} C_VEL
LIN {X 0,Y 277.592,Z 468.775,A -85,B 0,C 180,E1 -17704.347,E2 -17704.347} C_VEL
LIN {X 0,Y 278.325,Z 478.982,A -85,B 0,C 180,E1 -17705.563,E2 -17705.563} C_VEL
LIN {X 0,Y 278.338,Z 490.561,A -85,B 0,C 180,E1 -17707.156,E2 -17707.156} C_VEL
LIN {X 0,Y 278.054,Z 495.481,A -85,B 0,C 180,E1 -17707.915,E2 -17707.915} C_VEL
LIN {X 0,Y 276.013,Z 505.072,A -85,B 0,C 180,E1 -17709.506,E2 -17709.506} C_VEL
LIN {X 0,Y 274.068,Z 514.2,A -85,B 0,C 180,E1 -17711.382,E2 -17711.382} C_VEL
LIN {X 0,Y 272.343,Z 522.512,A -85,B 0,C 180,E1 -17713.509,E2 -17713.509} C_VEL
LIN {X 0,Y 270.845,Z 529.471,A -85,B 0,C 180,E1 -17715.729,E2 -17715.729} C_VEL
LIN {X 0,Y 269.657,Z 535.085,A -85,B 0,C 180,E1 -17717.965,E2 -17717.965} C_VEL
LIN {X 0,Y 268.945,Z 539.538,A -85,B 0,C 180,E1 -17720.22,E2 -17720.22} C_VEL
LIN {X 0,Y 268.516,Z 542.928,A -85,B 0,C 180,E1 -17722.48,E2 -17722.48} C_VEL
LIN {X 0,Y 268.351,Z 545.042,A -85,B 0,C 180,E1 -17724.386,E2 -17724.386} C_VEL
LIN {X 0,Y 268.339,Z 546.823,A -85,B 0,C 180,E1 -17726.997,E2 -17726.997} C_VEL
LIN {X 0,Y 268.442,Z 547.338,A -85,B 0,C 180,E1 -17730,E2 -17730} C_VEL
LIN {X 0,Y 268.356,Z 546.996,A -85,B 0,C 180,E1 -17731.5,E2 -17731.5} C_VEL
LIN {X 0,Y 268.351,Z 546.239,A -85,B 0,C 180,E1 -17733.002,E2 -17733.002} C_VEL
LIN {X 0,Y 268.418,Z 543.722,A -85,B 0,C 180,E1 -17735.756,E2 -17735.756} C_VEL
LIN {X 0,Y 268.631,Z 540.141,A -85,B 0,C 180,E1 -17738.273,E2 -17738.273} C_VEL
LIN {X 0,Y 269.163,Z 535.783,A -85,B 0,C 180,E1 -17740.531,E2 -17740.531} C_VEL
LIN {X 0,Y 269.941,Z 530.213,A -85,B 0,C 180,E1 -17742.785,E2 -17742.785} C_VEL
LIN {X 0,Y 271.208,Z 523.271,A -85,B 0,C 180,E1 -17745.018,E2 -17745.018} C_VEL
LIN {X 0,Y 272.711,Z 514.933,A -85,B 0,C 180,E1 -17747.151,E2 -17747.151} C_VEL
LIN {X 0,Y 274.172,Z 505.627,A -85,B 0,C 180,E1 -17749.076,E2 -17749.076} C_VEL
LIN {X 0,Y 275.881,Z 495.864,A -85,B 0,C 180,E1 -17750.698,E2 -17750.698} C_VEL
LIN {X 0,Y 276.633,Z 490.801,A -85,B 0,C 180,E1 -17751.419,E2 -17751.419} C_VEL
LIN {X 0,Y 276.011,Z 478.783,A -85,B 0,C 180,E1 -17752.993,E2 -17752.993} C_VEL
LIN {X 0,Y 274.908,Z 466.734,A -85,B 0,C 180,E1 -17754.278,E2 -17754.278} C_VEL
LIN {X 0,Y 272.954,Z 453.586,A -85,B 0,C 180,E1 -17755.419,E2 -17755.419} C_VEL
LIN {X 0,Y 270.407,Z 440.085,A -85,B 0,C 180,E1 -17756.324,E2 -17756.324} C_VEL
LIN {X 0,Y 271.357,Z 434.108,A -85,B 0,C 180,E1 -17760.333,E2 -17760.333} C_VEL
LIN {X 0,Y 272.526,Z 427.933,A -85,B 0,C 180,E1 -17764.564,E2 -17764.564} C_VEL
LIN {X 0,Y 273.101,Z 424.384,A -85,B 0,C 180,E1 -17767.084,E2 -17767.084} C_VEL
LIN {X 0,Y 272.665,Z 420.388,A -85,B 0,C 180,E1 -17770.118,E2 -17770.118} C_VEL
LIN {X 0,Y 271.768,Z 415.223,A -85,B 0,C 180,E1 -17774.283,E2 -17774.283} C_VEL
LIN {X 0,Y 270.792,Z 410.012,A -85,B 0,C 180,E1 -17778.819,E2 -17778.819} C_VEL
LIN {X 0,Y 270.238,Z 406.824,A -85,B 0,C 180,E1 -17781.855,E2 -17781.855} C_VEL
LIN {X 0,Y 270.21,Z 406.828,A -85,B 0,C 180,E1 -17785.096,E2 -17785.096} C_VEL
LIN {X 0,Y 270.195,Z 406.831,A -85,B 0,C 180,E1 -17789.13,E2 -17789.13} C_VEL
LIN {X 0,Y 270.259,Z 406.82,A -85,B 0,C 180,E1 -17792.145,E2 -17792.145} C_VEL
LIN {X 0,Y 270.271,Z 406.817,A -85,B 0,C 180,E1 -17795.519,E2 -17795.519} C_VEL
LIN {X 0,Y 270.296,Z 406.815,A -85,B 0,C 180,E1 -17800.244,E2 -17800.244} C_VEL
LIN {X 0,Y 270.396,Z 406.804,A -85,B 0,C 180,E1 -17804.935,E2 -17804.935} C_VEL
LIN {X 0,Y 270.406,Z 406.8,A -85,B 0,C 180,E1 -17809.518,E2 -17809.518} C_VEL
LIN {X 0,Y 270.592,Z 406.779,A -85,B 0,C 180,E1 -17812.538,E2 -17812.538} C_VEL
LIN {X 0,Y 270.781,Z 406.756,A -85,B 0,C 180,E1 -17818.513,E2 -17818.513} C_VEL
LIN {X 0,Y 270.781,Z 406.75,A -85,B 0,C 180,E1 -17821.487,E2 -17821.487} C_VEL
LIN {X 0,Y 270.604,Z 406.775,A -85,B 0,C 180,E1 -17827.462,E2 -17827.462} C_VEL
LIN {X 0,Y 270.435,Z 406.798,A -85,B 0,C 180,E1 -17830.481,E2 -17830.481} C_VEL
LIN {X 0,Y 270.39,Z 406.801,A -85,B 0,C 180,E1 -17835.066,E2 -17835.066} C_VEL
LIN {X 0,Y 270.296,Z 406.813,A -85,B 0,C 180,E1 -17839.756,E2 -17839.756} C_VEL
LIN {X 0,Y 270.269,Z 406.818,A -85,B 0,C 180,E1 -17844.586,E2 -17844.586} C_VEL
LIN {X 0,Y 270.267,Z 406.818,A -85,B 0,C 180,E1 -17847.909,E2 -17847.909} C_VEL
LIN {X 0,Y 270.18,Z 406.824,A -85,B 0,C 180,E1 -17851.349,E2 -17851.349} C_VEL
LIN {X 0,Y 270.211,Z 406.824,A -85,B 0,C 180,E1 -17854.904,E2 -17854.904} C_VEL
LIN {X 0,Y 270.219,Z 406.823,A -85,B 0,C 180,E1 -17858.718,E2 -17858.718} C_VEL
LIN {X 0,Y 270.182,Z 406.829,A -85,B 0,C 180,E1 -17862.557,E2 -17862.557} C_VEL
LIN {X 0,Y 270.163,Z 406.83,A -85,B 0,C 180,E1 -17866.752,E2 -17866.752} C_VEL
LIN {X 0,Y 270.196,Z 406.816,A -85,B 0,C 180,E1 -17871.291,E2 -17871.291} C_VEL
LIN {X 0,Y 270.201,Z 406.821,A -85,B 0,C 180,E1 -17875.096,E2 -17875.096} C_VEL
LIN {X 0,Y 270.2,Z 406.827,A -85,B 0,C 180,E1 -17879.132,E2 -17879.132} C_VEL
LIN {X 0,Y 270.264,Z 406.816,A -85,B 0,C 180,E1 -17882.147,E2 -17882.147} C_VEL
LIN {X 0,Y 270.278,Z 406.81,A -85,B 0,C 180,E1 -17885.52,E2 -17885.52} C_VEL
LIN {X 0,Y 270.303,Z 406.813,A -85,B 0,C 180,E1 -17890.245,E2 -17890.245} C_VEL
LIN {X 0,Y 270.405,Z 406.8,A -85,B 0,C 180,E1 -17894.936,E2 -17894.936} C_VEL
LIN {X 0,Y 270.444,Z 406.794,A -85,B 0,C 180,E1 -17899.52,E2 -17899.52} C_VEL
LIN {X 0,Y 270.615,Z 406.775,A -85,B 0,C 180,E1 -17902.539,E2 -17902.539} C_VEL
LIN {X 0,Y 270.713,Z 406.762,A -85,B 0,C 180,E1 -17908.513,E2 -17908.513} C_VEL
LIN {X 0,Y 270.043,Z 406.849,A -85,B 0,C 180,E1 -17910,E2 -17910} C_VEL
LIN {X 0,Y 269.688,Z 407.52,A -85,B 0,C 180,E1 -17911.494,E2 -17911.494} C_VEL
LIN {X 0,Y 269.749,Z 410.326,A -85,B 0,C 180,E1 -17915.232,E2 -17915.232} C_VEL
LIN {X 0,Y 269.707,Z 410.873,A -85,B 0,C 180,E1 -17915.936,E2 -17915.936} C_VEL
LIN {X 0,Y 274.054,Z 425.578,A -85,B 0,C 180,E1 -17917.182,E2 -17917.182} C_VEL
LIN {X 0,Y 277.076,Z 437.553,A -85,B 0,C 180,E1 -17918.413,E2 -17918.413} C_VEL
LIN {X 0,Y 279.078,Z 448.848,A -85,B 0,C 180,E1 -17919.787,E2 -17919.787} C_VEL
LIN {X 0,Y 277.524,Z 460.971,A -85,B 0,C 180,E1 -17921.318,E2 -17921.318} C_VEL
LIN {X 0,Y 275.797,Z 471.897,A -85,B 0,C 180,E1 -17923.071,E2 -17923.071} C_VEL
LIN {X 0,Y 274.261,Z 480.783,A -85,B 0,C 180,E1 -17924.848,E2 -17924.848} C_VEL
LIN {X 0,Y 272.746,Z 489.108,A -85,B 0,C 180,E1 -17926.896,E2 -17926.896} C_VEL
LIN {X 0,Y 271.516,Z 495.651,A -85,B 0,C 180,E1 -17928.878,E2 -17928.878} C_VEL
LIN {X 0,Y 270.333,Z 502.141,A -85,B 0,C 180,E1 -17931.344,E2 -17931.344} C_VEL
LIN {X 0,Y 269.411,Z 507.52,A -85,B 0,C 180,E1 -17934.072,E2 -17934.072} C_VEL
LIN {X 0,Y 268.918,Z 510.833,A -85,B 0,C 180,E1 -17936.377,E2 -17936.377} C_VEL
LIN {X 0,Y 268.561,Z 512.663,A -85,B 0,C 180,E1 -17938.102,E2 -17938.102} C_VEL
LIN {X 0,Y 268.334,Z 514.102,A -85,B 0,C 180,E1 -17940.195,E2 -17940.195} C_VEL
LIN {X 0,Y 268.323,Z 514.828,A -85,B 0,C 180,E1 -17943.053,E2 -17943.053} C_VEL
LIN {X 0,Y 268.619,Z 514.16,A -85,B 0,C 180,E1 -17945.799,E2 -17945.799} C_VEL
LIN {X 0,Y 269.317,Z 511.954,A -85,B 0,C 180,E1 -17948.777,E2 -17948.777} C_VEL
LIN {X 0,Y 270.269,Z 508.158,A -85,B 0,C 180,E1 -17951.672,E2 -17951.672} C_VEL
LIN {X 0,Y 271.536,Z 503.144,A -85,B 0,C 180,E1 -17954.332,E2 -17954.332} C_VEL
LIN {X 0,Y 273.037,Z 497.328,A -85,B 0,C 180,E1 -17956.648,E2 -17956.648} C_VEL
LIN {X 0,Y 274.866,Z 489.806,A -85,B 0,C 180,E1 -17958.981,E2 -17958.981} C_VEL
LIN {X 0,Y 276.845,Z 481.414,A -85,B 0,C 180,E1 -17961.051,E2 -17961.051} C_VEL
LIN {X 0,Y 278.627,Z 472.963,A -85,B 0,C 180,E1 -17962.744,E2 -17962.744} C_VEL
LIN {X 0,Y 280.66,Z 462.197,A -85,B 0,C 180,E1 -17964.471,E2 -17964.471} C_VEL
LIN {X 0,Y 282.05,Z 454.208,A -85,B 0,C 180,E1 -17965.517,E2 -17965.517} C_VEL
LIN {X 0,Y 281.829,Z 450.776,A -85,B 0,C 180,E1 -17965.994,E2 -17965.994} C_VEL
LIN {X 0,Y 279.186,Z 438.892,A -85,B 0,C 180,E1 -17967.661,E2 -17967.661} C_VEL
LIN {X 0,Y 275.394,Z 426.684,A -85,B 0,C 180,E1 -17969.203,E2 -17969.203} C_VEL
LIN {X 0,Y 270.932,Z 416.177,A -85,B 0,C 180,E1 -17970.471,E2 -17970.471} C_VEL
LIN {X 0,Y 270.083,Z 413.557,A -85,B 0,C 180,E1 -17970.743,E2 -17970.743} C_VEL
LIN {X 0,Y 270.262,Z 411.658,A -85,B 0,C 180,E1 -17973.763,E2 -17973.763} C_VEL
LIN {X 0,Y 270.42,Z 409.693,A -85,B 0,C 180,E1 -17977.055,E2 -17977.055} C_VEL
LIN {X 0,Y 270.404,Z 407.91,A -85,B 0,C 180,E1 -17980.252,E2 -17980.252} C_VEL
LIN {X 0,Y 270.338,Z 407.091,A -85,B 0,C 180,E1 -17981.822,E2 -17981.822} C_VEL
LIN {X 0,Y 270.394,Z 406.806,A -85,B 0,C 180,E1 -17984.935,E2 -17984.935} C_VEL
LIN {X 0,Y 270.41,Z 406.804,A -85,B 0,C 180,E1 -17989.518,E2 -17989.518} C_VEL
LIN {X 0,Y 270.595,Z 406.776,A -85,B 0,C 180,E1 -17992.538,E2 -17992.538} C_VEL
LIN {X 0,Y 270.784,Z 406.757,A -85,B 0,C 180,E1 -17998.513,E2 -17998.513} C_VEL
LIN {X 0,Y 270.785,Z 406.755,A -85,B 0,C 180,E1 -18001.487,E2 -18001.487} C_VEL
LIN {X 0,Y 270.595,Z 406.775,A -85,B 0,C 180,E1 -18007.461,E2 -18007.461} C_VEL
LIN {X 0,Y 270.41,Z 406.797,A -85,B 0,C 180,E1 -18010.482,E2 -18010.482} C_VEL
LIN {X 0,Y 270.393,Z 406.804,A -85,B 0,C 180,E1 -18015.065,E2 -18015.065} C_VEL
LIN {X 0,Y 270.344,Z 406.805,A -85,B 0,C 180,E1 -18016.674,E2 -18016.674} C_VEL
LIN {X 0,Y 269.577,Z 406.905,A -85,B 0,C 180,E1 -18017.917,E2 -18017.917} C_VEL
LIN {X 0,Y 266.631,Z 407.272,A -85,B 0,C 180,E1 -18019.942,E2 -18019.942} C_VEL
LIN {X 0,Y 264.21,Z 407.575,A -85,B 0,C 180,E1 -18021.589,E2 -18021.589} C_VEL
LIN {X 0,Y 263.218,Z 407.699,A -85,B 0,C 180,E1 -18022.866,E2 -18022.866} C_VEL
LIN {X 0,Y 263.159,Z 407.703,A -85,B 0,C 180,E1 -18023.299,E2 -18023.299} C_VEL
LIN {X 0,Y 263.188,Z 407.699,A -85,B 0,C 180,E1 -18026.998,E2 -18026.998} C_VEL
LIN {X 0,Y 263.162,Z 407.882,A -85,B 0,C 180,E1 -18031.287,E2 -18031.287} C_VEL
LIN {X 0,Y 263.593,Z 409.826,A -85,B 0,C 180,E1 -18034.257,E2 -18034.257} C_VEL
LIN {X 0,Y 264.033,Z 412.426,A -85,B 0,C 180,E1 -18037.75,E2 -18037.75} C_VEL
LIN {X 0,Y 264.598,Z 416.001,A -85,B 0,C 180,E1 -18041.952,E2 -18041.952} C_VEL
LIN {X 0,Y 265.404,Z 420.375,A -85,B 0,C 180,E1 -18046.49,E2 -18046.49} C_VEL
LIN {X 0,Y 266.12,Z 424.121,A -85,B 0,C 180,E1 -18049.984,E2 -18049.984} C_VEL
LIN {X 0,Y 266.344,Z 427.226,A -85,B 0,C 180,E1 -18052.635,E2 -18052.635} C_VEL
LIN {X 0,Y 265.781,Z 430.329,A -85,B 0,C 180,E1 -18055.058,E2 -18055.058} C_VEL
LIN {X 0,Y 264.454,Z 436.567,A -85,B 0,C 180,E1 -18059.673,E2 -18059.673} C_VEL
LIN {X 0,Y 264.219,Z 437.581,A -85,B 0,C 180,E1 -18060.401,E2 -18060.401} C_VEL
LIN {X 0,Y 265.163,Z 441.108,A -85,B 0,C 180,E1 -18060.702,E2 -18060.702} C_VEL
LIN {X 0,Y 268.508,Z 453.864,A -85,B 0,C 180,E1 -18061.963,E2 -18061.963} C_VEL
LIN {X 0,Y 270.706,Z 466.293,A -85,B 0,C 180,E1 -18063.314,E2 -18063.314} C_VEL
LIN {X 0,Y 271.683,Z 477.052,A -85,B 0,C 180,E1 -18064.626,E2 -18064.626} C_VEL
LIN {X 0,Y 271.792,Z 488.206,A -85,B 0,C 180,E1 -18066.17,E2 -18066.17} C_VEL
LIN {X 0,Y 271.485,Z 495.591,A -85,B 0,C 180,E1 -18067.352,E2 -18067.352} C_VEL
LIN {X 0,Y 269.361,Z 505.084,A -85,B 0,C 180,E1 -18068.976,E2 -18068.976} C_VEL
LIN {X 0,Y 267.329,Z 514.136,A -85,B 0,C 180,E1 -18070.895,E2 -18070.895} C_VEL
LIN {X 0,Y 265.533,Z 522.357,A -85,B 0,C 180,E1 -18073.074,E2 -18073.074} C_VEL
LIN {X 0,Y 263.928,Z 529.264,A -85,B 0,C 180,E1 -18075.347,E2 -18075.347} C_VEL
LIN {X 0,Y 262.668,Z 534.832,A -85,B 0,C 180,E1 -18077.64,E2 -18077.64} C_VEL
LIN {X 0,Y 261.904,Z 539.236,A -85,B 0,C 180,E1 -18079.955,E2 -18079.955} C_VEL
LIN {X 0,Y 261.437,Z 542.583,A -85,B 0,C 180,E1 -18082.275,E2 -18082.275} C_VEL
LIN {X 0,Y 261.251,Z 544.862,A -85,B 0,C 180,E1 -18084.472,E2 -18084.472} C_VEL
LIN {X 0,Y 261.268,Z 546.413,A -85,B 0,C 180,E1 -18086.916,E2 -18086.916} C_VEL
LIN {X 0,Y 261.356,Z 546.898,A -85,B 0,C 180,E1 -18090,E2 -18090} C_VEL
LIN {X 0,Y 261.277,Z 546.54,A -85,B 0,C 180,E1 -18091.541,E2 -18091.541} C_VEL
LIN {X 0,Y 261.283,Z 545.751,A -85,B 0,C 180,E1 -18093.083,E2 -18093.083} C_VEL
LIN {X 0,Y 261.338,Z 543.42,A -85,B 0,C 180,E1 -18095.722,E2 -18095.722} C_VEL
LIN {X 0,Y 261.576,Z 539.581,A -85,B 0,C 180,E1 -18098.497,E2 -18098.497} C_VEL
LIN {X 0,Y 262.127,Z 535.182,A -85,B 0,C 180,E1 -18100.817,E2 -18100.817} C_VEL
LIN {X 0,Y 262.962,Z 529.571,A -85,B 0,C 180,E1 -18103.13,E2 -18103.13} C_VEL
LIN {X 0,Y 264.278,Z 522.57,A -85,B 0,C 180,E1 -18105.422,E2 -18105.422} C_VEL
LIN {X 0,Y 265.781,Z 514.632,A -85,B 0,C 180,E1 -18107.498,E2 -18107.498} C_VEL
LIN {X 0,Y 267.417,Z 504.79,A -85,B 0,C 180,E1 -18109.577,E2 -18109.577} C_VEL
LIN {X 0,Y 269.257,Z 494.954,A -85,B 0,C 180,E1 -18111.232,E2 -18111.232} C_VEL
LIN {X 0,Y 269.691,Z 491.112,A -85,B 0,C 180,E1 -18111.798,E2 -18111.798} C_VEL
LIN {X 0,Y 269.173,Z 479.401,A -85,B 0,C 180,E1 -18113.401,E2 -18113.401} C_VEL
LIN {X 0,Y 268.016,Z 466.702,A -85,B 0,C 180,E1 -18114.806,E2 -18114.806} C_VEL
LIN {X 0,Y 266.059,Z 453.524,A -85,B 0,C 180,E1 -18115.992,E2 -18115.992} C_VEL
LIN {X 0,Y 263.463,Z 439.678,A -85,B 0,C 180,E1 -18116.966,E2 -18116.966} C_VEL
LIN {X 0,Y 264.472,Z 433.748,A -85,B 0,C 180,E1 -18121.072,E2 -18121.072} C_VEL
LIN {X 0,Y 265.747,Z 427.408,A -85,B 0,C 180,E1 -18125.577,E2 -18125.577} C_VEL
LIN {X 0,Y 266.028,Z 424.686,A -85,B 0,C 180,E1 -18127.576,E2 -18127.576} C_VEL
LIN {X 0,Y 265.691,Z 421.719,A -85,B 0,C 180,E1 -18129.906,E2 -18129.906} C_VEL
LIN {X 0,Y 264.898,Z 417.194,A -85,B 0,C 180,E1 -18133.613,E2 -18133.613} C_VEL
LIN {X 0,Y 264.076,Z 413.024,A -85,B 0,C 180,E1 -18137.263,E2 -18137.263} C_VEL
LIN {X 0,Y 263.474,Z 409.353,A -85,B 0,C 180,E1 -18140.672,E2 -18140.672} C_VEL
LIN {X 0,Y 263.194,Z 407.701,A -85,B 0,C 180,E1 -18142.424,E2 -18142.424} C_VEL
LIN {X 0,Y 263.179,Z 407.701,A -85,B 0,C 180,E1 -18145.89,E2 -18145.89} C_VEL
LIN {X 0,Y 263.145,Z 407.707,A -85,B 0,C 180,E1 -18149.506,E2 -18149.506} C_VEL
LIN {X 0,Y 263.186,Z 407.703,A -85,B 0,C 180,E1 -18153.002,E2 -18153.002} C_VEL
LIN {X 0,Y 263.178,Z 407.702,A -85,B 0,C 180,E1 -18156.387,E2 -18156.387} C_VEL
LIN {X 0,Y 263.258,Z 407.69,A -85,B 0,C 180,E1 -18159.693,E2 -18159.693} C_VEL
LIN {X 0,Y 263.345,Z 407.682,A -85,B 0,C 180,E1 -18164.522,E2 -18164.522} C_VEL
LIN {X 0,Y 263.349,Z 407.68,A -85,B 0,C 180,E1 -18169.233,E2 -18169.233} C_VEL
LIN {X 0,Y 263.551,Z 407.655,A -85,B 0,C 180,E1 -18172.338,E2 -18172.338} C_VEL
LIN {X 0,Y 263.745,Z 407.632,A -85,B 0,C 180,E1 -18178.473,E2 -18178.473} C_VEL
LIN {X 0,Y 263.746,Z 407.627,A -85,B 0,C 180,E1 -18181.527,E2 -18181.527} C_VEL
LIN {X 0,Y 263.566,Z 407.652,A -85,B 0,C 180,E1 -18187.662,E2 -18187.662} C_VEL
LIN {X 0,Y 263.368,Z 407.676,A -85,B 0,C 180,E1 -18190.766,E2 -18190.766} C_VEL
LIN {X 0,Y 263.339,Z 407.678,A -85,B 0,C 180,E1 -18195.479,E2 -18195.479} C_VEL
LIN {X 0,Y 263.258,Z 407.693,A -85,B 0,C 180,E1 -18200.307,E2 -18200.307} C_VEL
LIN {X 0,Y 263.204,Z 407.695,A -85,B 0,C 180,E1 -18205.292,E2 -18205.292} C_VEL
LIN {X 0,Y 263.175,Z 407.701,A -85,B 0,C 180,E1 -18208.73,E2 -18208.73} C_VEL
LIN {X 0,Y 263.129,Z 407.704,A -85,B 0,C 180,E1 -18212.289,E2 -18212.289} C_VEL
LIN {X 0,Y 263.185,Z 407.701,A -85,B 0,C 180,E1 -18215.979,E2 -18215.979} C_VEL
LIN {X 0,Y 263.135,Z 407.706,A -85,B 0,C 180,E1 -18219.868,E2 -18219.868} C_VEL
LIN {X 0,Y 263.124,Z 407.709,A -85,B 0,C 180,E1 -18223.984,E2 -18223.984} C_VEL
LIN {X 0,Y 263.122,Z 407.705,A -85,B 0,C 180,E1 -18228.408,E2 -18228.408} C_VEL
LIN {X 0,Y 263.18,Z 407.687,A -85,B 0,C 180,E1 -18233.238,E2 -18233.238} C_VEL
LIN {X 0,Y 263.132,Z 407.708,A -85,B 0,C 180,E1 -18237.713,E2 -18237.713} C_VEL
LIN {X 0,Y 263.196,Z 407.7,A -85,B 0,C 180,E1 -18241.786,E2 -18241.786} C_VEL
LIN {X 0,Y 263.227,Z 407.686,A -85,B 0,C 180,E1 -18245.201,E2 -18245.201} C_VEL
LIN {X 0,Y 263.265,Z 407.693,A -85,B 0,C 180,E1 -18249.694,E2 -18249.694} C_VEL
LIN {X 0,Y 263.353,Z 407.679,A -85,B 0,C 180,E1 -18254.523,E2 -18254.523} C_VEL
LIN {X 0,Y 263.377,Z 407.673,A -85,B 0,C 180,E1 -18259.235,E2 -18259.235} C_VEL
LIN {X 0,Y 263.576,Z 407.652,A -85,B 0,C 180,E1 -18262.339,E2 -18262.339} C_VEL
LIN {X 0,Y 263.673,Z 407.64,A -85,B 0,C 180,E1 -18268.473,E2 -18268.473} C_VEL
LIN {X 0,Y 262.979,Z 407.729,A -85,B 0,C 180,E1 -18270,E2 -18270} C_VEL
LIN {X 0,Y 262.657,Z 409.64,A -85,B 0,C 180,E1 -18273.068,E2 -18273.068} C_VEL
LIN {X 0,Y 262.723,Z 411.379,A -85,B 0,C 180,E1 -18275.324,E2 -18275.324} C_VEL
LIN {X 0,Y 266.679,Z 424.314,A -85,B 0,C 180,E1 -18276.431,E2 -18276.431} C_VEL
LIN {X 0,Y 269.667,Z 436.16,A -85,B 0,C 180,E1 -18277.657,E2 -18277.657} C_VEL
LIN {X 0,Y 271.787,Z 446.567,A -85,B 0,C 180,E1 -18278.926,E2 -18278.926} C_VEL
LIN {X 0,Y 272.29,Z 449.216,A -85,B 0,C 180,E1 -18279.284,E2 -18279.284} C_VEL
LIN {X 0,Y 271.213,Z 458.48,A -85,B 0,C 180,E1 -18280.451,E2 -18280.451} C_VEL
LIN {X 0,Y 269.425,Z 469.945,A -85,B 0,C 180,E1 -18282.236,E2 -18282.236} C_VEL
LIN {X 0,Y 267.736,Z 479.468,A -85,B 0,C 180,E1 -18284.087,E2 -18284.087} C_VEL
LIN {X 0,Y 266.126,Z 487.804,A -85,B 0,C 180,E1 -18286.099,E2 -18286.099} C_VEL
LIN {X 0,Y 264.549,Z 496.018,A -85,B 0,C 180,E1 -18288.59,E2 -18288.59} C_VEL
LIN {X 0,Y 263.393,Z 502.142,A -85,B 0,C 180,E1 -18290.95,E2 -18290.95} C_VEL
LIN {X 0,Y 262.438,Z 507.526,A -85,B 0,C 180,E1 -18293.684,E2 -18293.684} C_VEL
LIN {X 0,Y 261.847,Z 511.239,A -85,B 0,C 180,E1 -18296.287,E2 -18296.287} C_VEL
LIN {X 0,Y 261.342,Z 513.768,A -85,B 0,C 180,E1 -18298.95,E2 -18298.95} C_VEL
LIN {X 0,Y 261.224,Z 514.767,A -85,B 0,C 180,E1 -18300.742,E2 -18300.742} C_VEL
LIN {X 0,Y 261.261,Z 515.247,A -85,B 0,C 180,E1 -18303.497,E2 -18303.497} C_VEL
LIN {X 0,Y 261.638,Z 514.449,A -85,B 0,C 180,E1 -18306.307,E2 -18306.307} C_VEL
LIN {X 0,Y 262.306,Z 512.426,A -85,B 0,C 180,E1 -18309.013,E2 -18309.013} C_VEL
LIN {X 0,Y 263.276,Z 508.837,A -85,B 0,C 180,E1 -18311.863,E2 -18311.863} C_VEL
LIN {X 0,Y 264.316,Z 504.876,A -85,B 0,C 180,E1 -18314.117,E2 -18314.117} C_VEL
LIN {X 0,Y 265.892,Z 499.179,A -85,B 0,C 180,E1 -18316.589,E2 -18316.589} C_VEL
LIN {X 0,Y 267.747,Z 492.09,A -85,B 0,C 180,E1 -18318.988,E2 -18318.988} C_VEL
LIN {X 0,Y 269.524,Z 485.1,A -85,B 0,C 180,E1 -18320.872,E2 -18320.872} C_VEL
LIN {X 0,Y 271.479,Z 476.562,A -85,B 0,C 180,E1 -18322.754,E2 -18322.754} C_VEL
LIN {X 0,Y 273.514,Z 466.865,A -85,B 0,C 180,E1 -18324.474,E2 -18324.474} C_VEL
LIN {X 0,Y 275.64,Z 455.338,A -85,B 0,C 180,E1 -18326.099,E2 -18326.099} C_VEL
LIN {X 0,Y 274.44,Z 447.81,A -85,B 0,C 180,E1 -18327.249,E2 -18327.249} C_VEL
LIN {X 0,Y 272.073,Z 437.909,A -85,B 0,C 180,E1 -18328.666,E2 -18328.666} C_VEL
LIN {X 0,Y 268.474,Z 427.003,A -85,B 0,C 180,E1 -18330.119,E2 -18330.119} C_VEL
LIN {X 0,Y 264.226,Z 417.134,A -85,B 0,C 180,E1 -18331.394,E2 -18331.394} C_VEL
LIN {X 0,Y 263.122,Z 414.077,A -85,B 0,C 180,E1 -18331.758,E2 -18331.758} C_VEL
LIN {X 0,Y 263.338,Z 412.043,A -85,B 0,C 180,E1 -18335.147,E2 -18335.147} C_VEL
LIN {X 0,Y 263.458,Z 409.868,A -85,B 0,C 180,E1 -18339.011,E2 -18339.011} C_VEL
LIN {X 0,Y 263.296,Z 407.895,A -85,B 0,C 180,E1 -18342.925,E2 -18342.925} C_VEL
LIN {X 0,Y 263.302,Z 407.69,A -85,B 0,C 180,E1 -18346.1,E2 -18346.1} C_VEL
LIN {X 0,Y 263.469,Z 407.665,A -85,B 0,C 180,E1 -18350.79,E2 -18350.79} C_VEL
LIN {X 0,Y 263.506,Z 407.663,A -85,B 0,C 180,E1 -18353.876,E2 -18353.876} C_VEL
LIN {X 0,Y 263.748,Z 407.633,A -85,B 0,C 180,E1 -18358.473,E2 -18358.473} C_VEL
LIN {X 0,Y 263.749,Z 407.631,A -85,B 0,C 180,E1 -18361.527,E2 -18361.527} C_VEL
LIN {X 0,Y 263.555,Z 407.651,A -85,B 0,C 180,E1 -18367.662,E2 -18367.662} C_VEL
LIN {X 0,Y 263.352,Z 407.676,A -85,B 0,C 180,E1 -18370.766,E2 -18370.766} C_VEL
LIN {X 0,Y 263.342,Z 407.679,A -85,B 0,C 180,E1 -18375.478,E2 -18375.478} C_VEL
LIN {X 0,Y 263.261,Z 407.693,A -85,B 0,C 180,E1 -18380.307,E2 -18380.307} C_VEL
LIN {X 0,Y 263.159,Z 407.703,A -85,B 0,C 180,E1 -18383.299,E2 -18383.299} C_VEL
LIN {X 0,Y 262.532,Z 407.806,A -85,B 0,C 180,E1 -18384.579,E2 -18384.579} C_VEL
LIN {X 0,Y 259.642,Z 408.139,A -85,B 0,C 180,E1 -18386.664,E2 -18386.664} C_VEL
LIN {X 0,Y 257.191,Z 408.447,A -85,B 0,C 180,E1 -18388.357,E2 -18388.357} C_VEL
LIN {X 0,Y 256.183,Z 408.703,A -85,B 0,C 180,E1 -18389.668,E2 -18389.668} C_VEL
LIN {X 0,Y 256.126,Z 408.902,A -85,B 0,C 180,E1 -18390.109,E2 -18390.109} C_VEL
LIN {X 0,Y 256.525,Z 410.779,A -85,B 0,C 180,E1 -18393.226,E2 -18393.226} C_VEL
LIN {X 0,Y 257.079,Z 413.841,A -85,B 0,C 180,E1 -18397.553,E2 -18397.553} C_VEL
LIN {X 0,Y 257.48,Z 416.589,A -85,B 0,C 180,E1 -18400.926,E2 -18400.926} C_VEL
LIN {X 0,Y 258.18,Z 420.345,A -85,B 0,C 180,E1 -18405.052,E2 -18405.052} C_VEL
LIN {X 0,Y 259.023,Z 424.804,A -85,B 0,C 180,E1 -18409.439,E2 -18409.439} C_VEL
LIN {X 0,Y 259.273,Z 427.476,A -85,B 0,C 180,E1 -18411.822,E2 -18411.822} C_VEL
LIN {X 0,Y 259.222,Z 429.314,A -85,B 0,C 180,E1 -18413.383,E2 -18413.383} C_VEL
LIN {X 0,Y 257.958,Z 434.779,A -85,B 0,C 180,E1 -18417.628,E2 -18417.628} C_VEL
LIN {X 0,Y 257.477,Z 437.059,A -85,B 0,C 180,E1 -18419.354,E2 -18419.354} C_VEL
LIN {X 0,Y 258.474,Z 440.805,A -85,B 0,C 180,E1 -18419.704,E2 -18419.704} C_VEL
LIN {X 0,Y 261.897,Z 453.496,A -85,B 0,C 180,E1 -18421.038,E2 -18421.038} C_VEL
LIN {X 0,Y 264.088,Z 465.78,A -85,B 0,C 180,E1 -18422.45,E2 -18422.45} C_VEL
LIN {X 0,Y 265.135,Z 476.818,A -85,B 0,C 180,E1 -18423.856,E2 -18423.856} C_VEL
LIN {X 0,Y 265.245,Z 487.173,A -85,B 0,C 180,E1 -18425.335,E2 -18425.335} C_VEL
LIN {X 0,Y 264.704,Z 496.96,A -85,B 0,C 180,E1 -18426.945,E2 -18426.945} C_VEL
LIN {X 0,Y 262.303,Z 507.005,A -85,B 0,C 180,E1 -18428.795,E2 -18428.795} C_VEL
LIN {X 0,Y 259.954,Z 516.777,A -85,B 0,C 180,E1 -18431.069,E2 -18431.069} C_VEL
LIN {X 0,Y 258.39,Z 523.45,A -85,B 0,C 180,E1 -18432.999,E2 -18432.999} C_VEL
LIN {X 0,Y 257.042,Z 529.059,A -85,B 0,C 180,E1 -18434.945,E2 -18434.945} C_VEL
LIN {X 0,Y 255.694,Z 534.581,A -85,B 0,C 180,E1 -18437.297,E2 -18437.297} C_VEL
LIN {X 0,Y 254.867,Z 538.941,A -85,B 0,C 180,E1 -18439.674,E2 -18439.674} C_VEL
LIN {X 0,Y 254.374,Z 542.249,A -85,B 0,C 180,E1 -18442.059,E2 -18442.059} C_VEL
LIN {X 0,Y 254.175,Z 544.635,A -85,B 0,C 180,E1 -18444.507,E2 -18444.507} C_VEL
LIN {X 0,Y 254.175,Z 546.004,A -85,B 0,C 180,E1 -18446.83,E2 -18446.83} C_VEL
LIN {X 0,Y 254.179,Z 546.424,A -85,B 0,C 180,E1 -18448.415,E2 -18448.415} C_VEL
LIN {X 0,Y 254.272,Z 546.455,A -85,B 0,C 180,E1 -18450,E2 -18450} C_VEL
LIN {X 0,Y 254.2,Z 546.078,A -85,B 0,C 180,E1 -18451.584,E2 -18451.584} C_VEL
LIN {X 0,Y 254.214,Z 545.257,A -85,B 0,C 180,E1 -18453.169,E2 -18453.169} C_VEL
LIN {X 0,Y 254.243,Z 543.151,A -85,B 0,C 180,E1 -18455.648,E2 -18455.648} C_VEL
LIN {X 0,Y 254.397,Z 540.261,A -85,B 0,C 180,E1 -18457.939,E2 -18457.939} C_VEL
LIN {X 0,Y 254.893,Z 536.194,A -85,B 0,C 180,E1 -18460.324,E2 -18460.324} C_VEL
LIN {X 0,Y 255.844,Z 529.925,A -85,B 0,C 180,E1 -18463.098,E2 -18463.098} C_VEL
LIN {X 0,Y 257.167,Z 523.107,A -85,B 0,C 180,E1 -18465.453,E2 -18465.453} C_VEL
LIN {X 0,Y 258.783,Z 514.737,A -85,B 0,C 180,E1 -18467.757,E2 -18467.757} C_VEL
LIN {X 0,Y 260.342,Z 505.853,A -85,B 0,C 180,E1 -18469.72,E2 -18469.72} C_VEL
LIN {X 0,Y 262.132,Z 496.299,A -85,B 0,C 180,E1 -18471.425,E2 -18471.425} C_VEL
LIN {X 0,Y 262.764,Z 491.334,A -85,B 0,C 180,E1 -18472.196,E2 -18472.196} C_VEL
LIN {X 0,Y 262.309,Z 479.803,A -85,B 0,C 180,E1 -18473.84,E2 -18473.84} C_VEL
LIN {X 0,Y 261.331,Z 468.248,A -85,B 0,C 180,E1 -18475.193,E2 -18475.193} C_VEL
LIN {X 0,Y 259.499,Z 455.267,A -85,B 0,C 180,E1 -18476.437,E2 -18476.437} C_VEL
LIN {X 0,Y 256.999,Z 441.884,A -85,B 0,C 180,E1 -18477.453,E2 -18477.453} C_VEL
LIN {X 0,Y 256.537,Z 439.217,A -85,B 0,C 180,E1 -18477.667,E2 -18477.667} C_VEL
LIN {X 0,Y 257.688,Z 432.801,A -85,B 0,C 180,E1 -18482.277,E2 -18482.277} C_VEL
LIN {X 0,Y 258.634,Z 428.532,A -85,B 0,C 180,E1 -18485.392,E2 -18485.392} C_VEL
LIN {X 0,Y 258.972,Z 424.999,A -85,B 0,C 180,E1 -18488.094,E2 -18488.094} C_VEL
LIN {X 0,Y 258.329,Z 420.612,A -85,B 0,C 180,E1 -18491.684,E2 -18491.684} C_VEL
LIN {X 0,Y 257.567,Z 416.568,A -85,B 0,C 180,E1 -18495.188,E2 -18495.188} C_VEL
LIN {X 0,Y 256.604,Z 411.306,A -85,B 0,C 180,E1 -18500.072,E2 -18500.072} C_VEL
LIN {X 0,Y 256.164,Z 408.577,A -85,B 0,C 180,E1 -18502.873,E2 -18502.873} C_VEL
LIN {X 0,Y 256.08,Z 408.588,A -85,B 0,C 180,E1 -18506.709,E2 -18506.709} C_VEL
LIN {X 0,Y 256.132,Z 408.581,A -85,B 0,C 180,E1 -18511.405,E2 -18511.405} C_VEL
LIN {X 0,Y 256.161,Z 408.574,A -85,B 0,C 180,E1 -18515.699,E2 -18515.699} C_VEL
LIN {X 0,Y 256.161,Z 408.577,A -85,B 0,C 180,E1 -18519.105,E2 -18519.105} C_VEL
LIN {X 0,Y 256.294,Z 408.558,A -85,B 0,C 180,E1 -18524.085,E2 -18524.085} C_VEL
LIN {X 0,Y 256.291,Z 408.561,A -85,B 0,C 180,E1 -18528.933,E2 -18528.933} C_VEL
LIN {X 0,Y 256.509,Z 408.531,A -85,B 0,C 180,E1 -18532.126,E2 -18532.126} C_VEL
LIN {X 0,Y 256.493,Z 408.535,A -85,B 0,C 180,E1 -18536.859,E2 -18536.859} C_VEL
LIN {X 0,Y 256.767,Z 408.499,A -85,B 0,C 180,E1 -18540,E2 -18540} C_VEL
LIN {X 0,Y 256.493,Z 408.527,A -85,B 0,C 180,E1 -18543.142,E2 -18543.142} C_VEL
LIN {X 0,Y 256.534,Z 408.528,A -85,B 0,C 180,E1 -18547.873,E2 -18547.873} C_VEL
LIN {X 0,Y 256.303,Z 408.554,A -85,B 0,C 180,E1 -18551.067,E2 -18551.067} C_VEL
LIN {X 0,Y 256.289,Z 408.557,A -85,B 0,C 180,E1 -18555.916,E2 -18555.916} C_VEL
LIN {X 0,Y 256.161,Z 408.572,A -85,B 0,C 180,E1 -18560.896,E2 -18560.896} C_VEL
LIN {X 0,Y 256.184,Z 408.57,A -85,B 0,C 180,E1 -18565.139,E2 -18565.139} C_VEL
LIN {X 0,Y 256.11,Z 408.58,A -85,B 0,C 180,E1 -18569.601,E2 -18569.601} C_VEL
LIN {X 0,Y 256.081,Z 408.579,A -85,B 0,C 180,E1 -18573.291,E2 -18573.291} C_VEL
LIN {X 0,Y 256.137,Z 408.577,A -85,B 0,C 180,E1 -18577.279,E2 -18577.279} C_VEL
LIN {X 0,Y 256.07,Z 408.58,A -85,B 0,C 180,E1 -18581.201,E2 -18581.201} C_VEL
LIN {X 0,Y 256.057,Z 408.588,A -85,B 0,C 180,E1 -18585.531,E2 -18585.531} C_VEL
LIN {X 0,Y 256.052,Z 408.583,A -85,B 0,C 180,E1 -18588.798,E2 -18588.798} C_VEL
LIN {X 0,Y 256.129,Z 408.565,A -85,B 0,C 180,E1 -18592.868,E2 -18592.868} C_VEL
LIN {X 0,Y 256.067,Z 408.587,A -85,B 0,C 180,E1 -18596.708,E2 -18596.708} C_VEL
LIN {X 0,Y 256.104,Z 408.583,A -85,B 0,C 180,E1 -18600.4,E2 -18600.4} C_VEL
LIN {X 0,Y 256.189,Z 408.562,A -85,B 0,C 180,E1 -18604.862,E2 -18604.862} C_VEL
LIN {X 0,Y 256.168,Z 408.574,A -85,B 0,C 180,E1 -18609.106,E2 -18609.106} C_VEL
LIN {X 0,Y 256.302,Z 408.557,A -85,B 0,C 180,E1 -18614.086,E2 -18614.086} C_VEL
LIN {X 0,Y 256.312,Z 408.552,A -85,B 0,C 180,E1 -18618.935,E2 -18618.935} C_VEL
LIN {X 0,Y 256.544,Z 408.53,A -85,B 0,C 180,E1 -18622.128,E2 -18622.128} C_VEL
LIN {X 0,Y 256.264,Z 408.562,A -85,B 0,C 180,E1 -18625.281,E2 -18625.281} C_VEL
LIN {X 0,Y 256.609,Z 408.52,A -85,B 0,C 180,E1 -18628.431,E2 -18628.431} C_VEL
LIN {X 0,Y 255.915,Z 408.609,A -85,B 0,C 180,E1 -18630,E2 -18630} C_VEL
LIN {X 0,Y 255.74,Z 411.7,A -85,B 0,C 180,E1 -18634.631,E2 -18634.631} C_VEL
LIN {X 0,Y 260.317,Z 426.786,A -85,B 0,C 180,E1 -18636.005,E2 -18636.005} C_VEL
LIN {X 0,Y 263.108,Z 438.139,A -85,B 0,C 180,E1 -18637.251,E2 -18637.251} C_VEL
LIN {X 0,Y 265.14,Z 448.41,A -85,B 0,C 180,E1 -18638.574,E2 -18638.574} C_VEL
LIN {X 0,Y 265.557,Z 450.992,A -85,B 0,C 180,E1 -18638.945,E2 -18638.945} C_VEL
LIN {X 0,Y 264.051,Z 461.888,A -85,B 0,C 180,E1 -18640.405,E2 -18640.405} C_VEL
LIN {X 0,Y 262.273,Z 472.482,A -85,B 0,C 180,E1 -18642.182,E2 -18642.182} C_VEL
LIN {X 0,Y 260.607,Z 481.416,A -85,B 0,C 180,E1 -18644.047,E2 -18644.047} C_VEL
LIN {X 0,Y 258.959,Z 489.626,A -85,B 0,C 180,E1 -18646.152,E2 -18646.152} C_VEL
LIN {X 0,Y 257.601,Z 496.368,A -85,B 0,C 180,E1 -18648.284,E2 -18648.284} C_VEL
LIN {X 0,Y 256.317,Z 502.9,A -85,B 0,C 180,E1 -18650.882,E2 -18650.882} C_VEL
LIN {X 0,Y 255.39,Z 507.917,A -85,B 0,C 180,E1 -18653.517,E2 -18653.517} C_VEL
LIN {X 0,Y 254.788,Z 511.642,A -85,B 0,C 180,E1 -18656.189,E2 -18656.189} C_VEL
LIN {X 0,Y 254.401,Z 513.494,A -85,B 0,C 180,E1 -18658.011,E2 -18658.011} C_VEL
LIN {X 0,Y 254.131,Z 515.27,A -85,B 0,C 180,E1 -18660.984,E2 -18660.984} C_VEL
LIN {X 0,Y 254.239,Z 515.667,A -85,B 0,C 180,E1 -18663.972,E2 -18663.972} C_VEL
LIN {X 0,Y 254.66,Z 514.739,A -85,B 0,C 180,E1 -18666.838,E2 -18666.838} C_VEL
LIN {X 0,Y 255.416,Z 512.553,A -85,B 0,C 180,E1 -18669.606,E2 -18669.606} C_VEL
LIN {X 0,Y 256.342,Z 509.259,A -85,B 0,C 180,E1 -18672.247,E2 -18672.247} C_VEL
LIN {X 0,Y 257.816,Z 504.147,A -85,B 0,C 180,E1 -18675.133,E2 -18675.133} C_VEL
LIN {X 0,Y 259.587,Z 498.097,A -85,B 0,C 180,E1 -18677.665,E2 -18677.665} C_VEL
LIN {X 0,Y 261.339,Z 491.63,A -85,B 0,C 180,E1 -18679.803,E2 -18679.803} C_VEL
LIN {X 0,Y 263.707,Z 482.489,A -85,B 0,C 180,E1 -18682.195,E2 -18682.195} C_VEL
LIN {X 0,Y 265.958,Z 472.919,A -85,B 0,C 180,E1 -18684.178,E2 -18684.178} C_VEL
LIN {X 0,Y 268.239,Z 462.044,A -85,B 0,C 180,E1 -18685.953,E2 -18685.953} C_VEL
LIN {X 0,Y 269.219,Z 456.268,A -85,B 0,C 180,E1 -18686.755,E2 -18686.755} C_VEL
LIN {X 0,Y 267.238,Z 445.446,A -85,B 0,C 180,E1 -18688.487,E2 -18688.487} C_VEL
LIN {X 0,Y 264.382,Z 434.977,A -85,B 0,C 180,E1 -18690.021,E2 -18690.021} C_VEL
LIN {X 0,Y 259.976,Z 423.426,A -85,B 0,C 180,E1 -18691.65,E2 -18691.65} C_VEL
LIN {X 0,Y 257.162,Z 417.421,A -85,B 0,C 180,E1 -18692.481,E2 -18692.481} C_VEL
LIN {X 0,Y 256.19,Z 414.624,A -85,B 0,C 180,E1 -18692.811,E2 -18692.811} C_VEL
LIN {X 0,Y 256.35,Z 412.952,A -85,B 0,C 180,E1 -18695.717,E2 -18695.717} C_VEL
LIN {X 0,Y 256.479,Z 411.109,A -85,B 0,C 180,E1 -18699.131,E2 -18699.131} C_VEL
LIN {X 0,Y 256.338,Z 408.726,A -85,B 0,C 180,E1 -18704.087,E2 -18704.087} C_VEL
LIN {X 0,Y 256.294,Z 408.559,A -85,B 0,C 180,E1 -18708.933,E2 -18708.933} C_VEL
LIN {X 0,Y 256.512,Z 408.531,A -85,B 0,C 180,E1 -18712.126,E2 -18712.126} C_VEL
LIN {X 0,Y 256.496,Z 408.532,A -85,B 0,C 180,E1 -18716.858,E2 -18716.858} C_VEL
LIN {X 0,Y 256.762,Z 408.498,A -85,B 0,C 180,E1 -18720,E2 -18720} C_VEL
LIN {X 0,Y 256.496,Z 408.533,A -85,B 0,C 180,E1 -18723.141,E2 -18723.141} C_VEL
LIN {X 0,Y 256.512,Z 408.528,A -85,B 0,C 180,E1 -18727.874,E2 -18727.874} C_VEL
LIN {X 0,Y 256.29,Z 408.558,A -85,B 0,C 180,E1 -18732.672,E2 -18732.672} C_VEL
LIN {X 0,Y 256.276,Z 408.557,A -85,B 0,C 180,E1 -18736.299,E2 -18736.299} C_VEL
LIN {X 0,Y 256.155,Z 408.577,A -85,B 0,C 180,E1 -18741.12,E2 -18741.12} C_VEL
LIN {X 0,Y 256.186,Z 408.575,A -85,B 0,C 180,E1 -18745.138,E2 -18745.138} C_VEL
LIN {X 0,Y 256.101,Z 408.614,A -85,B 0,C 180,E1 -18749.601,E2 -18749.601} C_VEL
LIN {X 0,Y 256.126,Z 408.902,A -85,B 0,C 180,E1 -18750.109,E2 -18750.109} C_VEL
LIN {X 0,Y 255.593,Z 409.821,A -85,B 0,C 180,E1 -18751.41,E2 -18751.41} C_VEL
LIN {X 0,Y 253.059,Z 411.822,A -85,B 0,C 180,E1 -18753.522,E2 -18753.522} C_VEL
LIN {X 0,Y 250.916,Z 413.534,A -85,B 0,C 180,E1 -18755.235,E2 -18755.235} C_VEL
LIN {X 0,Y 250.065,Z 414.706,A -85,B 0,C 180,E1 -18756.562,E2 -18756.562} C_VEL
LIN {X 0,Y 250.035,Z 415.048,A -85,B 0,C 180,E1 -18757.012,E2 -18757.012} C_VEL
LIN {X 0,Y 250.525,Z 417.97,A -85,B 0,C 180,E1 -18760.762,E2 -18760.762} C_VEL
LIN {X 0,Y 251.099,Z 421.169,A -85,B 0,C 180,E1 -18764.405,E2 -18764.405} C_VEL
LIN {X 0,Y 251.933,Z 425.503,A -85,B 0,C 180,E1 -18768.868,E2 -18768.868} C_VEL
LIN {X 0,Y 252.236,Z 429.113,A -85,B 0,C 180,E1 -18772.195,E2 -18772.195} C_VEL
LIN {X 0,Y 251.979,Z 431.408,A -85,B 0,C 180,E1 -18774.147,E2 -18774.147} C_VEL
LIN {X 0,Y 250.718,Z 436.533,A -85,B 0,C 180,E1 -18778.218,E2 -18778.218} C_VEL
LIN {X 0,Y 251.671,Z 440.036,A -85,B 0,C 180,E1 -18778.575,E2 -18778.575} C_VEL
LIN {X 0,Y 255.393,Z 453.425,A -85,B 0,C 180,E1 -18780.094,E2 -18780.094} C_VEL
LIN {X 0,Y 257.597,Z 465.831,A -85,B 0,C 180,E1 -18781.59,E2 -18781.59} C_VEL
LIN {X 0,Y 258.701,Z 477.677,A -85,B 0,C 180,E1 -18783.189,E2 -18783.189} C_VEL
LIN {X 0,Y 258.656,Z 488.773,A -85,B 0,C 180,E1 -18784.878,E2 -18784.878} C_VEL
LIN {X 0,Y 258.165,Z 497.132,A -85,B 0,C 180,E1 -18786.326,E2 -18786.326} C_VEL
LIN {X 0,Y 255.693,Z 507.056,A -85,B 0,C 180,E1 -18788.219,E2 -18788.219} C_VEL
LIN {X 0,Y 253.212,Z 516.747,A -85,B 0,C 180,E1 -18790.545,E2 -18790.545} C_VEL
LIN {X 0,Y 251.601,Z 523.351,A -85,B 0,C 180,E1 -18792.526,E2 -18792.526} C_VEL
LIN {X 0,Y 250.177,Z 528.886,A -85,B 0,C 180,E1 -18794.521,E2 -18794.521} C_VEL
LIN {X 0,Y 248.73,Z 534.343,A -85,B 0,C 180,E1 -18796.936,E2 -18796.936} C_VEL
LIN {X 0,Y 247.847,Z 538.649,A -85,B 0,C 180,E1 -18799.379,E2 -18799.379} C_VEL
LIN {X 0,Y 247.332,Z 541.918,A -85,B 0,C 180,E1 -18801.832,E2 -18801.832} C_VEL
LIN {X 0,Y 247.088,Z 544.43,A -85,B 0,C 180,E1 -18804.572,E2 -18804.572} C_VEL
LIN {X 0,Y 247.085,Z 545.596,A -85,B 0,C 180,E1 -18806.738,E2 -18806.738} C_VEL
LIN {X 0,Y 247.105,Z 546,A -85,B 0,C 180,E1 -18808.37,E2 -18808.37} C_VEL
LIN {X 0,Y 247.191,Z 546.012,A -85,B 0,C 180,E1 -18810,E2 -18810} C_VEL
LIN {X 0,Y 247.126,Z 545.606,A -85,B 0,C 180,E1 -18811.629,E2 -18811.629} C_VEL
LIN {X 0,Y 247.147,Z 544.756,A -85,B 0,C 180,E1 -18813.26,E2 -18813.26} C_VEL
LIN {X 0,Y 247.164,Z 542.828,A -85,B 0,C 180,E1 -18815.609,E2 -18815.609} C_VEL
LIN {X 0,Y 247.353,Z 539.676,A -85,B 0,C 180,E1 -18818.167,E2 -18818.167} C_VEL
LIN {X 0,Y 247.863,Z 535.561,A -85,B 0,C 180,E1 -18820.62,E2 -18820.62} C_VEL
LIN {X 0,Y 248.874,Z 529.24,A -85,B 0,C 180,E1 -18823.472,E2 -18823.472} C_VEL
LIN {X 0,Y 250.251,Z 522.364,A -85,B 0,C 180,E1 -18825.891,E2 -18825.891} C_VEL
LIN {X 0,Y 251.872,Z 514.359,A -85,B 0,C 180,E1 -18828.142,E2 -18828.142} C_VEL
LIN {X 0,Y 253.613,Z 504.932,A -85,B 0,C 180,E1 -18830.266,E2 -18830.266} C_VEL
LIN {X 0,Y 255.715,Z 494.114,A -85,B 0,C 180,E1 -18832.203,E2 -18832.203} C_VEL
LIN {X 0,Y 255.674,Z 484.481,A -85,B 0,C 180,E1 -18833.703,E2 -18833.703} C_VEL
LIN {X 0,Y 254.871,Z 472.241,A -85,B 0,C 180,E1 -18835.301,E2 -18835.301} C_VEL
LIN {X 0,Y 253.468,Z 460.214,A -85,B 0,C 180,E1 -18836.593,E2 -18836.593} C_VEL
LIN {X 0,Y 251.173,Z 446.761,A -85,B 0,C 180,E1 -18837.759,E2 -18837.759} C_VEL
LIN {X 0,Y 249.617,Z 438.91,A -85,B 0,C 180,E1 -18838.312,E2 -18838.312} C_VEL
LIN {X 0,Y 250.744,Z 432.885,A -85,B 0,C 180,E1 -18842.769,E2 -18842.769} C_VEL
LIN {X 0,Y 251.687,Z 428.716,A -85,B 0,C 180,E1 -18845.925,E2 -18845.925} C_VEL
LIN {X 0,Y 251.904,Z 425.278,A -85,B 0,C 180,E1 -18848.631,E2 -18848.631} C_VEL
LIN {X 0,Y 251.178,Z 421.125,A -85,B 0,C 180,E1 -18852.183,E2 -18852.183} C_VEL
LIN {X 0,Y 250.489,Z 417.453,A -85,B 0,C 180,E1 -18855.458,E2 -18855.458} C_VEL
LIN {X 0,Y 249.692,Z 413.043,A -85,B 0,C 180,E1 -18859.656,E2 -18859.656} C_VEL
LIN {X 0,Y 249.087,Z 409.458,A -85,B 0,C 180,E1 -18863.47,E2 -18863.47} C_VEL
LIN {X 0,Y 249.035,Z 409.465,A -85,B 0,C 180,E1 -18867.844,E2 -18867.844} C_VEL
LIN {X 0,Y 249.091,Z 409.459,A -85,B 0,C 180,E1 -18871.338,E2 -18871.338} C_VEL
LIN {X 0,Y 249.146,Z 409.451,A -85,B 0,C 180,E1 -18874.968,E2 -18874.968} C_VEL
LIN {X 0,Y 249.105,Z 409.454,A -85,B 0,C 180,E1 -18880.211,E2 -18880.211} C_VEL
LIN {X 0,Y 249.237,Z 409.437,A -85,B 0,C 180,E1 -18883.622,E2 -18883.622} C_VEL
LIN {X 0,Y 249.238,Z 409.44,A -85,B 0,C 180,E1 -18888.616,E2 -18888.616} C_VEL
LIN {X 0,Y 249.448,Z 409.41,A -85,B 0,C 180,E1 -18891.902,E2 -18891.902} C_VEL
LIN {X 0,Y 249.29,Z 409.428,A -85,B 0,C 180,E1 -18895.149,E2 -18895.149} C_VEL
LIN {X 0,Y 249.67,Z 409.385,A -85,B 0,C 180,E1 -18898.387,E2 -18898.387} C_VEL
LIN {X 0,Y 249.67,Z 409.38,A -85,B 0,C 180,E1 -18901.613,E2 -18901.613} C_VEL
LIN {X 0,Y 249.444,Z 409.411,A -85,B 0,C 180,E1 -18906.745,E2 -18906.745} C_VEL
LIN {X 0,Y 249.383,Z 409.418,A -85,B 0,C 180,E1 -18909.735,E2 -18909.735} C_VEL
LIN {X 0,Y 249.195,Z 409.442,A -85,B 0,C 180,E1 -18914.704,E2 -18914.704} C_VEL
LIN {X 0,Y 249.134,Z 409.452,A -85,B 0,C 180,E1 -18918.078,E2 -18918.078} C_VEL
LIN {X 0,Y 249.082,Z 409.452,A -85,B 0,C 180,E1 -18921.519,E2 -18921.519} C_VEL
LIN {X 0,Y 249.126,Z 409.449,A -85,B 0,C 180,E1 -18925.483,E2 -18925.483} C_VEL
LIN {X 0,Y 249.079,Z 409.456,A -85,B 0,C 180,E1 -18928.994,E2 -18928.994} C_VEL
LIN {X 0,Y 249.032,Z 409.459,A -85,B 0,C 180,E1 -18932.426,E2 -18932.426} C_VEL
LIN {X 0,Y 249.071,Z 409.461,A -85,B 0,C 180,E1 -18936.339,E2 -18936.339} C_VEL
LIN {X 0,Y 249.031,Z 409.458,A -85,B 0,C 180,E1 -18940.474,E2 -18940.474} C_VEL
LIN {X 0,Y 249.003,Z 409.467,A -85,B 0,C 180,E1 -18944.88,E2 -18944.88} C_VEL
LIN {X 0,Y 249.014,Z 409.464,A -85,B 0,C 180,E1 -18947.364,E2 -18947.364} C_VEL
LIN {X 0,Y 249.042,Z 409.445,A -85,B 0,C 180,E1 -18952.201,E2 -18952.201} C_VEL
LIN {X 0,Y 249.043,Z 409.457,A -85,B 0,C 180,E1 -18955.641,E2 -18955.641} C_VEL
LIN {X 0,Y 249.048,Z 409.464,A -85,B 0,C 180,E1 -18959.474,E2 -18959.474} C_VEL
LIN {X 0,Y 249.073,Z 409.452,A -85,B 0,C 180,E1 -18963.163,E2 -18963.163} C_VEL
LIN {X 0,Y 249.081,Z 409.455,A -85,B 0,C 180,E1 -18966.734,E2 -18966.734} C_VEL
LIN {X 0,Y 249.113,Z 409.453,A -85,B 0,C 180,E1 -18970.213,E2 -18970.213} C_VEL
LIN {X 0,Y 249.244,Z 409.431,A -85,B 0,C 180,E1 -18973.623,E2 -18973.623} C_VEL
LIN {X 0,Y 249.256,Z 409.431,A -85,B 0,C 180,E1 -18978.617,E2 -18978.617} C_VEL
LIN {X 0,Y 249.488,Z 409.41,A -85,B 0,C 180,E1 -18981.904,E2 -18981.904} C_VEL
LIN {X 0,Y 249.459,Z 409.41,A -85,B 0,C 180,E1 -18983.53,E2 -18983.53} C_VEL
LIN {X 0,Y 249.548,Z 409.4,A -85,B 0,C 180,E1 -18988.387,E2 -18988.387} C_VEL
LIN {X 0,Y 248.852,Z 409.489,A -85,B 0,C 180,E1 -18990,E2 -18990} C_VEL
LIN {X 0,Y 248.639,Z 412.114,A -85,B 0,C 180,E1 -18993.9,E2 -18993.9} C_VEL
LIN {X 0,Y 253.44,Z 427.275,A -85,B 0,C 180,E1 -18995.371,E2 -18995.371} C_VEL
LIN {X 0,Y 256.36,Z 439.33,A -85,B 0,C 180,E1 -18996.743,E2 -18996.743} C_VEL
LIN {X 0,Y 258.351,Z 449.15,A -85,B 0,C 180,E1 -18998.061,E2 -18998.061} C_VEL
LIN {X 0,Y 258.792,Z 452.603,A -85,B 0,C 180,E1 -18998.563,E2 -18998.563} C_VEL
LIN {X 0,Y 257.047,Z 463.992,A -85,B 0,C 180,E1 -19000.168,E2 -19000.168} C_VEL
LIN {X 0,Y 255.077,Z 474.925,A -85,B 0,C 180,E1 -19002.128,E2 -19002.128} C_VEL
LIN {X 0,Y 253.345,Z 483.819,A -85,B 0,C 180,E1 -19004.113,E2 -19004.113} C_VEL
LIN {X 0,Y 251.774,Z 491.447,A -85,B 0,C 180,E1 -19006.209,E2 -19006.209} C_VEL
LIN {X 0,Y 250.136,Z 499.081,A -85,B 0,C 180,E1 -19008.851,E2 -19008.851} C_VEL
LIN {X 0,Y 249.003,Z 505.082,A -85,B 0,C 180,E1 -19011.526,E2 -19011.526} C_VEL
LIN {X 0,Y 248.133,Z 509.531,A -85,B 0,C 180,E1 -19014.125,E2 -19014.125} C_VEL
LIN {X 0,Y 247.487,Z 513.038,A -85,B 0,C 180,E1 -19017.024,E2 -19017.024} C_VEL
LIN {X 0,Y 247.181,Z 514.598,A -85,B 0,C 180,E1 -19018.905,E2 -19018.905} C_VEL
LIN {X 0,Y 247.027,Z 515.826,A -85,B 0,C 180,E1 -19021.404,E2 -19021.404} C_VEL
LIN {X 0,Y 247.223,Z 516.048,A -85,B 0,C 180,E1 -19024.649,E2 -19024.649} C_VEL
LIN {X 0,Y 247.704,Z 514.985,A -85,B 0,C 180,E1 -19027.398,E2 -19027.398} C_VEL
LIN {X 0,Y 248.655,Z 512.346,A -85,B 0,C 180,E1 -19030.547,E2 -19030.547} C_VEL
LIN {X 0,Y 249.916,Z 508.109,A -85,B 0,C 180,E1 -19033.679,E2 -19033.679} C_VEL
LIN {X 0,Y 251.637,Z 502.521,A -85,B 0,C 180,E1 -19036.564,E2 -19036.564} C_VEL
LIN {X 0,Y 253.554,Z 496.206,A -85,B 0,C 180,E1 -19039.052,E2 -19039.052} C_VEL
LIN {X 0,Y 255.859,Z 488.141,A -85,B 0,C 180,E1 -19041.52,E2 -19041.52} C_VEL
LIN {X 0,Y 258.217,Z 479.133,A -85,B 0,C 180,E1 -19043.704,E2 -19043.704} C_VEL
LIN {X 0,Y 260.379,Z 470.058,A -85,B 0,C 180,E1 -19045.471,E2 -19045.471} C_VEL
LIN {X 0,Y 262.63,Z 459.195,A -85,B 0,C 180,E1 -19047.156,E2 -19047.156} C_VEL
LIN {X 0,Y 262.589,Z 456.235,A -85,B 0,C 180,E1 -19047.636,E2 -19047.636} C_VEL
LIN {X 0,Y 260.43,Z 445.139,A -85,B 0,C 180,E1 -19049.481,E2 -19049.481} C_VEL
LIN {X 0,Y 257.574,Z 435.022,A -85,B 0,C 180,E1 -19051.044,E2 -19051.044} C_VEL
LIN {X 0,Y 252.739,Z 422.814,A -85,B 0,C 180,E1 -19052.873,E2 -19052.873} C_VEL
LIN {X 0,Y 250.509,Z 418.44,A -85,B 0,C 180,E1 -19053.553,E2 -19053.553} C_VEL
LIN {X 0,Y 249.314,Z 415.489,A -85,B 0,C 180,E1 -19053.946,E2 -19053.946} C_VEL
LIN {X 0,Y 249.244,Z 415.14,A -85,B 0,C 180,E1 -19054.035,E2 -19054.035} C_VEL
LIN {X 0,Y 249.458,Z 412.799,A -85,B 0,C 180,E1 -19058.388,E2 -19058.388} C_VEL
LIN {X 0,Y 249.362,Z 411.104,A -85,B 0,C 180,E1 -19061.939,E2 -19061.939} C_VEL
LIN {X 0,Y 249.227,Z 409.633,A -85,B 0,C 180,E1 -19065.298,E2 -19065.298} C_VEL
LIN {X 0,Y 249.242,Z 409.437,A -85,B 0,C 180,E1 -19068.616,E2 -19068.616} C_VEL
LIN {X 0,Y 249.452,Z 409.412,A -85,B 0,C 180,E1 -19071.902,E2 -19071.902} C_VEL
LIN {X 0,Y 249.293,Z 409.429,A -85,B 0,C 180,E1 -19075.148,E2 -19075.148} C_VEL
LIN {X 0,Y 249.673,Z 409.386,A -85,B 0,C 180,E1 -19078.387,E2 -19078.387} C_VEL
LIN {X 0,Y 249.673,Z 409.384,A -85,B 0,C 180,E1 -19081.613,E2 -19081.613} C_VEL
LIN {X 0,Y 249.45,Z 409.414,A -85,B 0,C 180,E1 -19086.471,E2 -19086.471} C_VEL
LIN {X 0,Y 249.341,Z 409.425,A -85,B 0,C 180,E1 -19089.736,E2 -19089.736} C_VEL
LIN {X 0,Y 249.198,Z 409.444,A -85,B 0,C 180,E1 -19094.704,E2 -19094.704} C_VEL
LIN {X 0,Y 249.136,Z 409.449,A -85,B 0,C 180,E1 -19098.077,E2 -19098.077} C_VEL
LIN {X 0,Y 249.085,Z 409.459,A -85,B 0,C 180,E1 -19101.518,E2 -19101.518} C_VEL
LIN {X 0,Y 249.128,Z 409.454,A -85,B 0,C 180,E1 -19105.482,E2 -19105.482} C_VEL
LIN {X 0,Y 249.128,Z 409.815,A -85,B 0,C 180,E1 -19108.658,E2 -19108.658} C_VEL
LIN {X 0,Y 249.498,Z 411.896,A -85,B 0,C 180,E1 -19112.358,E2 -19112.358} C_VEL
LIN {X 0,Y 249.974,Z 414.447,A -85,B 0,C 180,E1 -19116.186,E2 -19116.186} C_VEL
LIN {X 0,Y 250.035,Z 415.048,A -85,B 0,C 180,E1 -19117.012,E2 -19117.012} C_VEL
LIN {X 0,Y 249.547,Z 416.184,A -85,B 0,C 180,E1 -19118.335,E2 -19118.335} C_VEL
LIN {X 0,Y 247.062,Z 418.499,A -85,B 0,C 180,E1 -19120.484,E2 -19120.484} C_VEL
LIN {X 0,Y 244.939,Z 420.454,A -85,B 0,C 180,E1 -19122.227,E2 -19122.227} C_VEL
LIN {X 0,Y 244.097,Z 421.836,A -85,B 0,C 180,E1 -19123.576,E2 -19123.576} C_VEL
LIN {X 0,Y 244.068,Z 422.261,A -85,B 0,C 180,E1 -19124.033,E2 -19124.033} C_VEL
LIN {X 0,Y 244.834,Z 426.226,A -85,B 0,C 180,E1 -19128.274,E2 -19128.274} C_VEL
LIN {X 0,Y 245.204,Z 428.904,A -85,B 0,C 180,E1 -19130.909,E2 -19130.909} C_VEL
LIN {X 0,Y 245.131,Z 431.672,A -85,B 0,C 180,E1 -19133.396,E2 -19133.396} C_VEL
LIN {X 0,Y 244.012,Z 436.012,A -85,B 0,C 180,E1 -19137.011,E2 -19137.011} C_VEL
LIN {X 0,Y 244.954,Z 439.5,A -85,B 0,C 180,E1 -19137.384,E2 -19137.384} C_VEL
LIN {X 0,Y 247.84,Z 449.124,A -85,B 0,C 180,E1 -19138.538,E2 -19138.538} C_VEL
LIN {X 0,Y 250.263,Z 460.043,A -85,B 0,C 180,E1 -19139.916,E2 -19139.916} C_VEL
LIN {X 0,Y 251.967,Z 473.116,A -85,B 0,C 180,E1 -19141.695,E2 -19141.695} C_VEL
LIN {X 0,Y 252.367,Z 483.686,A -85,B 0,C 180,E1 -19143.288,E2 -19143.288} C_VEL
LIN {X 0,Y 251.778,Z 495.132,A -85,B 0,C 180,E1 -19145.247,E2 -19145.247} C_VEL
LIN {X 0,Y 251.197,Z 499.451,A -85,B 0,C 180,E1 -19146.066,E2 -19146.066} C_VEL
LIN {X 0,Y 248.632,Z 508.897,A -85,B 0,C 180,E1 -19148.005,E2 -19148.005} C_VEL
LIN {X 0,Y 246.11,Z 518.26,A -85,B 0,C 180,E1 -19150.452,E2 -19150.452} C_VEL
LIN {X 0,Y 244.142,Z 525.543,A -85,B 0,C 180,E1 -19152.839,E2 -19152.839} C_VEL
LIN {X 0,Y 242.247,Z 532.476,A -85,B 0,C 180,E1 -19155.723,E2 -19155.723} C_VEL
LIN {X 0,Y 241.141,Z 537.1,A -85,B 0,C 180,E1 -19158.228,E2 -19158.228} C_VEL
LIN {X 0,Y 240.421,Z 540.657,A -85,B 0,C 180,E1 -19160.748,E2 -19160.748} C_VEL
LIN {X 0,Y 240.081,Z 543.227,A -85,B 0,C 180,E1 -19163.275,E2 -19163.275} C_VEL
LIN {X 0,Y 239.989,Z 544.414,A -85,B 0,C 180,E1 -19164.96,E2 -19164.96} C_VEL
LIN {X 0,Y 239.998,Z 545.191,A -85,B 0,C 180,E1 -19166.642,E2 -19166.642} C_VEL
LIN {X 0,Y 240.032,Z 545.576,A -85,B 0,C 180,E1 -19168.322,E2 -19168.322} C_VEL
LIN {X 0,Y 240.112,Z 545.57,A -85,B 0,C 180,E1 -19170,E2 -19170} C_VEL
LIN {X 0,Y 240.054,Z 545.126,A -85,B 0,C 180,E1 -19171.677,E2 -19171.677} C_VEL
LIN {X 0,Y 240.058,Z 544.255,A -85,B 0,C 180,E1 -19173.356,E2 -19173.356} C_VEL
LIN {X 0,Y 240.092,Z 542.487,A -85,B 0,C 180,E1 -19175.585,E2 -19175.585} C_VEL
LIN {X 0,Y 240.304,Z 539.089,A -85,B 0,C 180,E1 -19178.408,E2 -19178.408} C_VEL
LIN {X 0,Y 240.853,Z 534.927,A -85,B 0,C 180,E1 -19180.933,E2 -19180.933} C_VEL
LIN {X 0,Y 241.94,Z 528.557,A -85,B 0,C 180,E1 -19183.865,E2 -19183.865} C_VEL
LIN {X 0,Y 243.374,Z 521.623,A -85,B 0,C 180,E1 -19186.352,E2 -19186.352} C_VEL
LIN {X 0,Y 244.869,Z 514.537,A -85,B 0,C 180,E1 -19188.403,E2 -19188.403} C_VEL
LIN {X 0,Y 246.543,Z 505.972,A -85,B 0,C 180,E1 -19190.438,E2 -19190.438} C_VEL
LIN {X 0,Y 248.694,Z 495.448,A -85,B 0,C 180,E1 -19192.426,E2 -19192.426} C_VEL
LIN {X 0,Y 248.934,Z 490.409,A -85,B 0,C 180,E1 -19193.281,E2 -19193.281} C_VEL
LIN {X 0,Y 248.491,Z 478.914,A -85,B 0,C 180,E1 -19195.015,E2 -19195.015} C_VEL
LIN {X 0,Y 247.533,Z 467.394,A -85,B 0,C 180,E1 -19196.446,E2 -19196.446} C_VEL
LIN {X 0,Y 245.631,Z 453.948,A -85,B 0,C 180,E1 -19197.816,E2 -19197.816} C_VEL
LIN {X 0,Y 243.198,Z 441.09,A -85,B 0,C 180,E1 -19198.86,E2 -19198.86} C_VEL
LIN {X 0,Y 242.721,Z 438.434,A -85,B 0,C 180,E1 -19199.077,E2 -19199.077} C_VEL
LIN {X 0,Y 244.064,Z 431.841,A -85,B 0,C 180,E1 -19204.158,E2 -19204.158} C_VEL
LIN {X 0,Y 244.819,Z 428.129,A -85,B 0,C 180,E1 -19207.073,E2 -19207.073} C_VEL
LIN {X 0,Y 244.769,Z 425.629,A -85,B 0,C 180,E1 -19209.173,E2 -19209.173} C_VEL
LIN {X 0,Y 243.828,Z 420.308,A -85,B 0,C 180,E1 -19213.897,E2 -19213.897} C_VEL
LIN {X 0,Y 242.839,Z 415.193,A -85,B 0,C 180,E1 -19218.802,E2 -19218.802} C_VEL
LIN {X 0,Y 242.281,Z 411.603,A -85,B 0,C 180,E1 -19222.471,E2 -19222.471} C_VEL
LIN {X 0,Y 242.033,Z 410.338,A -85,B 0,C 180,E1 -19223.985,E2 -19223.985} C_VEL
LIN {X 0,Y 241.971,Z 410.346,A -85,B 0,C 180,E1 -19228.479,E2 -19228.479} C_VEL
LIN {X 0,Y 242.003,Z 410.341,A -85,B 0,C 180,E1 -19232.312,E2 -19232.312} C_VEL
LIN {X 0,Y 242.052,Z 410.332,A -85,B 0,C 180,E1 -19236.015,E2 -19236.015} C_VEL
LIN {X 0,Y 242.032,Z 410.335,A -85,B 0,C 180,E1 -19239.608,E2 -19239.608} C_VEL
LIN {X 0,Y 242.158,Z 410.32,A -85,B 0,C 180,E1 -19243.278,E2 -19243.278} C_VEL
LIN {X 0,Y 242.175,Z 410.318,A -85,B 0,C 180,E1 -19248.279,E2 -19248.279} C_VEL
LIN {X 0,Y 242.394,Z 410.288,A -85,B 0,C 180,E1 -19251.665,E2 -19251.665} C_VEL
LIN {X 0,Y 242.251,Z 410.305,A -85,B 0,C 180,E1 -19255.007,E2 -19255.007} C_VEL
LIN {X 0,Y 242.631,Z 410.262,A -85,B 0,C 180,E1 -19258.34,E2 -19258.34} C_VEL
LIN {X 0,Y 242.631,Z 410.256,A -85,B 0,C 180,E1 -19261.66,E2 -19261.66} C_VEL
LIN {X 0,Y 242.423,Z 410.288,A -85,B 0,C 180,E1 -19266.722,E2 -19266.722} C_VEL
LIN {X 0,Y 242.309,Z 410.3,A -85,B 0,C 180,E1 -19270.022,E2 -19270.022} C_VEL
LIN {X 0,Y 242.158,Z 410.317,A -85,B 0,C 180,E1 -19275.142,E2 -19275.142} C_VEL
LIN {X 0,Y 242.068,Z 410.332,A -85,B 0,C 180,E1 -19278.625,E2 -19278.625} C_VEL
LIN {X 0,Y 242.008,Z 410.333,A -85,B 0,C 180,E1 -19282.181,E2 -19282.181} C_VEL
LIN {X 0,Y 242.062,Z 410.329,A -85,B 0,C 180,E1 -19285.839,E2 -19285.839} C_VEL
LIN {X 0,Y 242.026,Z 410.334,A -85,B 0,C 180,E1 -19289.581,E2 -19289.581} C_VEL
LIN {X 0,Y 241.988,Z 410.335,A -85,B 0,C 180,E1 -19293.492,E2 -19293.492} C_VEL
LIN {X 0,Y 242.008,Z 410.338,A -85,B 0,C 180,E1 -19297.579,E2 -19297.579} C_VEL
LIN {X 0,Y 241.947,Z 410.34,A -85,B 0,C 180,E1 -19301.921,E2 -19301.921} C_VEL
LIN {X 0,Y 241.933,Z 410.347,A -85,B 0,C 180,E1 -19306.572,E2 -19306.572} C_VEL
LIN {X 0,Y 241.955,Z 410.333,A -85,B 0,C 180,E1 -19310.282,E2 -19310.282} C_VEL
LIN {X 0,Y 241.98,Z 410.334,A -85,B 0,C 180,E1 -19314.489,E2 -19314.489} C_VEL
LIN {X 0,Y 241.973,Z 410.346,A -85,B 0,C 180,E1 -19318.481,E2 -19318.481} C_VEL
LIN {X 0,Y 242.003,Z 410.334,A -85,B 0,C 180,E1 -19322.313,E2 -19322.313} C_VEL
LIN {X 0,Y 242.059,Z 410.326,A -85,B 0,C 180,E1 -19326.017,E2 -19326.017} C_VEL
LIN {X 0,Y 242.04,Z 410.336,A -85,B 0,C 180,E1 -19329.609,E2 -19329.609} C_VEL
LIN {X 0,Y 242.165,Z 410.31,A -85,B 0,C 180,E1 -19333.279,E2 -19333.279} C_VEL
LIN {X 0,Y 242.189,Z 410.312,A -85,B 0,C 180,E1 -19338.281,E2 -19338.281} C_VEL
LIN {X 0,Y 242.438,Z 410.288,A -85,B 0,C 180,E1 -19341.667,E2 -19341.667} C_VEL
LIN {X 0,Y 242.432,Z 410.286,A -85,B 0,C 180,E1 -19343.342,E2 -19343.342} C_VEL
LIN {X 0,Y 242.49,Z 410.279,A -85,B 0,C 180,E1 -19348.34,E2 -19348.34} C_VEL
LIN {X 0,Y 241.79,Z 410.368,A -85,B 0,C 180,E1 -19350,E2 -19350} C_VEL
LIN {X 0,Y 241.553,Z 412.599,A -85,B 0,C 180,E1 -19353.18,E2 -19353.18} C_VEL
LIN {X 0,Y 245.642,Z 424.786,A -85,B 0,C 180,E1 -19354.369,E2 -19354.369} C_VEL
LIN {X 0,Y 248.521,Z 435.668,A -85,B 0,C 180,E1 -19355.606,E2 -19355.606} C_VEL
LIN {X 0,Y 251.041,Z 447.109,A -85,B 0,C 180,E1 -19357.131,E2 -19357.131} C_VEL
LIN {X 0,Y 251.973,Z 454.539,A -85,B 0,C 180,E1 -19358.219,E2 -19358.219} C_VEL
LIN {X 0,Y 250.028,Z 466.107,A -85,B 0,C 180,E1 -19359.951,E2 -19359.951} C_VEL
LIN {X 0,Y 248.137,Z 476.2,A -85,B 0,C 180,E1 -19361.85,E2 -19361.85} C_VEL
LIN {X 0,Y 246.28,Z 485.377,A -85,B 0,C 180,E1 -19364.01,E2 -19364.01} C_VEL
LIN {X 0,Y 244.58,Z 493.116,A -85,B 0,C 180,E1 -19366.27,E2 -19366.27} C_VEL
LIN {X 0,Y 242.975,Z 500.522,A -85,B 0,C 180,E1 -19368.99,E2 -19368.99} C_VEL
LIN {X 0,Y 241.872,Z 506.023,A -85,B 0,C 180,E1 -19371.593,E2 -19371.593} C_VEL
LIN {X 0,Y 241.061,Z 510.086,A -85,B 0,C 180,E1 -19374.089,E2 -19374.089} C_VEL
LIN {X 0,Y 240.663,Z 512.427,A -85,B 0,C 180,E1 -19375.979,E2 -19375.979} C_VEL
LIN {X 0,Y 240.145,Z 514.807,A -85,B 0,C 180,E1 -19378.601,E2 -19378.601} C_VEL
LIN {X 0,Y 239.949,Z 516.383,A -85,B 0,C 180,E1 -19381.853,E2 -19381.853} C_VEL
LIN {X 0,Y 240.17,Z 516.455,A -85,B 0,C 180,E1 -19384.979,E2 -19384.979} C_VEL
LIN {X 0,Y 240.752,Z 515.23,A -85,B 0,C 180,E1 -19387.984,E2 -19387.984} C_VEL
LIN {X 0,Y 241.677,Z 512.818,A -85,B 0,C 180,E1 -19390.879,E2 -19390.879} C_VEL
LIN {X 0,Y 242.973,Z 508.832,A -85,B 0,C 180,E1 -19393.963,E2 -19393.963} C_VEL
LIN {X 0,Y 244.374,Z 504.564,A -85,B 0,C 180,E1 -19396.352,E2 -19396.352} C_VEL
LIN {X 0,Y 246.374,Z 498.401,A -85,B 0,C 180,E1 -19398.997,E2 -19398.997} C_VEL
LIN {X 0,Y 248.709,Z 490.744,A -85,B 0,C 180,E1 -19401.561,E2 -19401.561} C_VEL
LIN {X 0,Y 250.898,Z 483.142,A -85,B 0,C 180,E1 -19403.587,E2 -19403.587} C_VEL
LIN {X 0,Y 253.335,Z 473.69,A -85,B 0,C 180,E1 -19405.62,E2 -19405.62} C_VEL
LIN {X 0,Y 255.677,Z 463.597,A -85,B 0,C 180,E1 -19407.348,E2 -19407.348} C_VEL
LIN {X 0,Y 256.399,Z 459.359,A -85,B 0,C 180,E1 -19407.993,E2 -19407.993} C_VEL
LIN {X 0,Y 254.478,Z 448.33,A -85,B 0,C 180,E1 -19409.962,E2 -19409.962} C_VEL
LIN {X 0,Y 251.721,Z 438.066,A -85,B 0,C 180,E1 -19411.664,E2 -19411.664} C_VEL
LIN {X 0,Y 247.5,Z 426.838,A -85,B 0,C 180,E1 -19413.49,E2 -19413.49} C_VEL
LIN {X 0,Y 243.538,Z 418.819,A -85,B 0,C 180,E1 -19414.808,E2 -19414.808} C_VEL
LIN {X 0,Y 242.363,Z 415.723,A -85,B 0,C 180,E1 -19415.25,E2 -19415.25} C_VEL
LIN {X 0,Y 242.462,Z 414.279,A -85,B 0,C 180,E1 -19418.055,E2 -19418.055} C_VEL
LIN {X 0,Y 242.407,Z 412.709,A -85,B 0,C 180,E1 -19421.402,E2 -19421.402} C_VEL
LIN {X 0,Y 242.311,Z 411.243,A -85,B 0,C 180,E1 -19424.868,E2 -19424.868} C_VEL
LIN {X 0,Y 242.2,Z 410.574,A -85,B 0,C 180,E1 -19426.577,E2 -19426.577} C_VEL
LIN {X 0,Y 242.33,Z 410.297,A -85,B 0,C 180,E1 -19430.417,E2 -19430.417} C_VEL
LIN {X 0,Y 242.421,Z 410.288,A -85,B 0,C 180,E1 -19433.341,E2 -19433.341} C_VEL
LIN {X 0,Y 242.633,Z 410.263,A -85,B 0,C 180,E1 -19438.34,E2 -19438.34} C_VEL
LIN {X 0,Y 242.634,Z 410.26,A -85,B 0,C 180,E1 -19441.66,E2 -19441.66} C_VEL
LIN {X 0,Y 242.421,Z 410.289,A -85,B 0,C 180,E1 -19446.659,E2 -19446.659} C_VEL
LIN {X 0,Y 242.265,Z 410.304,A -85,B 0,C 180,E1 -19450.024,E2 -19450.024} C_VEL
LIN {X 0,Y 242.161,Z 410.319,A -85,B 0,C 180,E1 -19455.141,E2 -19455.141} C_VEL
LIN {X 0,Y 242.07,Z 410.326,A -85,B 0,C 180,E1 -19458.624,E2 -19458.624} C_VEL
LIN {X 0,Y 242.011,Z 410.339,A -85,B 0,C 180,E1 -19462.18,E2 -19462.18} C_VEL
LIN {X 0,Y 242.065,Z 410.33,A -85,B 0,C 180,E1 -19465.838,E2 -19465.838} C_VEL
LIN {X 0,Y 242.277,Z 411.995,A -85,B 0,C 180,E1 -19469.547,E2 -19469.547} C_VEL
LIN {X 0,Y 242.697,Z 414.197,A -85,B 0,C 180,E1 -19473.381,E2 -19473.381} C_VEL
LIN {X 0,Y 243.159,Z 416.884,A -85,B 0,C 180,E1 -19477.37,E2 -19477.37} C_VEL
LIN {X 0,Y 243.707,Z 420.134,A -85,B 0,C 180,E1 -19481.55,E2 -19481.55} C_VEL
LIN {X 0,Y 244.068,Z 422.261,A -85,B 0,C 180,E1 -19484.033,E2 -19484.033} C_VEL
LIN {X 0,Y 243.596,Z 423.615,A -85,B 0,C 180,E1 -19485.377,E2 -19485.377} C_VEL
LIN {X 0,Y 241.162,Z 426.206,A -85,B 0,C 180,E1 -19487.563,E2 -19487.563} C_VEL
LIN {X 0,Y 238.394,Z 429.422,A -85,B 0,C 180,E1 -19490.245,E2 -19490.245} C_VEL
LIN {X 0,Y 238.181,Z 430.42,A -85,B 0,C 180,E1 -19491.171,E2 -19491.171} C_VEL
LIN {X 0,Y 238.217,Z 432.141,A -85,B 0,C 180,E1 -19492.803,E2 -19492.803} C_VEL
LIN {X 0,Y 237.378,Z 435.489,A -85,B 0,C 180,E1 -19495.705,E2 -19495.705} C_VEL
LIN {X 0,Y 238.229,Z 438.828,A -85,B 0,C 180,E1 -19496.07,E2 -19496.07} C_VEL
LIN {X 0,Y 241.39,Z 448.964,A -85,B 0,C 180,E1 -19497.406,E2 -19497.406} C_VEL
LIN {X 0,Y 243.991,Z 460.652,A -85,B 0,C 180,E1 -19498.974,E2 -19498.974} C_VEL
LIN {X 0,Y 245.543,Z 472.77,A -85,B 0,C 180,E1 -19500.722,E2 -19500.722} C_VEL
LIN {X 0,Y 245.908,Z 484.491,A -85,B 0,C 180,E1 -19502.581,E2 -19502.581} C_VEL
LIN {X 0,Y 245.27,Z 495.451,A -85,B 0,C 180,E1 -19504.544,E2 -19504.544} C_VEL
LIN {X 0,Y 244.74,Z 499.7,A -85,B 0,C 180,E1 -19505.394,E2 -19505.394} C_VEL
LIN {X 0,Y 242.053,Z 508.998,A -85,B 0,C 180,E1 -19507.374,E2 -19507.374} C_VEL
LIN {X 0,Y 239.538,Z 517.726,A -85,B 0,C 180,E1 -19509.724,E2 -19509.724} C_VEL
LIN {X 0,Y 237.696,Z 524.302,A -85,B 0,C 180,E1 -19511.913,E2 -19511.913} C_VEL
LIN {X 0,Y 235.88,Z 530.47,A -85,B 0,C 180,E1 -19514.445,E2 -19514.445} C_VEL
LIN {X 0,Y 234.458,Z 535.417,A -85,B 0,C 180,E1 -19517.008,E2 -19517.008} C_VEL
LIN {X 0,Y 233.588,Z 539.269,A -85,B 0,C 180,E1 -19519.6,E2 -19519.6} C_VEL
LIN {X 0,Y 233.221,Z 541.285,A -85,B 0,C 180,E1 -19521.334,E2 -19521.334} C_VEL
LIN {X 0,Y 233.004,Z 542.883,A -85,B 0,C 180,E1 -19523.07,E2 -19523.07} C_VEL
LIN {X 0,Y 232.921,Z 544.033,A -85,B 0,C 180,E1 -19524.806,E2 -19524.806} C_VEL
LIN {X 0,Y 232.915,Z 544.788,A -85,B 0,C 180,E1 -19526.54,E2 -19526.54} C_VEL
LIN {X 0,Y 232.959,Z 545.153,A -85,B 0,C 180,E1 -19528.271,E2 -19528.271} C_VEL
LIN {X 0,Y 233.035,Z 545.122,A -85,B 0,C 180,E1 -19530,E2 -19530} C_VEL
LIN {X 0,Y 232.983,Z 544.638,A -85,B 0,C 180,E1 -19531.728,E2 -19531.728} C_VEL
LIN {X 0,Y 232.973,Z 543.744,A -85,B 0,C 180,E1 -19533.458,E2 -19533.458} C_VEL
LIN {X 0,Y 233.029,Z 542.108,A -85,B 0,C 180,E1 -19535.581,E2 -19535.581} C_VEL
LIN {X 0,Y 233.252,Z 538.483,A -85,B 0,C 180,E1 -19538.664,E2 -19538.664} C_VEL
LIN {X 0,Y 233.86,Z 534.27,A -85,B 0,C 180,E1 -19541.264,E2 -19541.264} C_VEL
LIN {X 0,Y 235.03,Z 527.843,A -85,B 0,C 180,E1 -19544.281,E2 -19544.281} C_VEL
LIN {X 0,Y 236.532,Z 520.827,A -85,B 0,C 180,E1 -19546.839,E2 -19546.839} C_VEL
LIN {X 0,Y 238.074,Z 513.661,A -85,B 0,C 180,E1 -19548.948,E2 -19548.948} C_VEL
LIN {X 0,Y 239.825,Z 504.973,A -85,B 0,C 180,E1 -19551.037,E2 -19551.037} C_VEL
LIN {X 0,Y 242.044,Z 494.33,A -85,B 0,C 180,E1 -19553.077,E2 -19553.077} C_VEL
LIN {X 0,Y 241.854,Z 482.95,A -85,B 0,C 180,E1 -19554.981,E2 -19554.981} C_VEL
LIN {X 0,Y 241.041,Z 470.543,A -85,B 0,C 180,E1 -19556.677,E2 -19556.677} C_VEL
LIN {X 0,Y 239.458,Z 458.036,A -85,B 0,C 180,E1 -19558.099,E2 -19558.099} C_VEL
LIN {X 0,Y 237.267,Z 445.301,A -85,B 0,C 180,E1 -19559.268,E2 -19559.268} C_VEL
LIN {X 0,Y 235.787,Z 438.045,A -85,B 0,C 180,E1 -19559.852,E2 -19559.852} C_VEL
LIN {X 0,Y 237.031,Z 432.459,A -85,B 0,C 180,E1 -19564.287,E2 -19564.287} C_VEL
LIN {X 0,Y 237.768,Z 429.063,A -85,B 0,C 180,E1 -19567.053,E2 -19567.053} C_VEL
LIN {X 0,Y 237.634,Z 425.921,A -85,B 0,C 180,E1 -19569.741,E2 -19569.741} C_VEL
LIN {X 0,Y 236.698,Z 420.725,A -85,B 0,C 180,E1 -19574.553,E2 -19574.553} C_VEL
LIN {X 0,Y 235.823,Z 416.196,A -85,B 0,C 180,E1 -19579.031,E2 -19579.031} C_VEL
LIN {X 0,Y 235.169,Z 412.197,A -85,B 0,C 180,E1 -19583.295,E2 -19583.295} C_VEL
LIN {X 0,Y 234.987,Z 411.215,A -85,B 0,C 180,E1 -19584.586,E2 -19584.586} C_VEL
LIN {X 0,Y 234.956,Z 411.22,A -85,B 0,C 180,E1 -19587.424,E2 -19587.424} C_VEL
LIN {X 0,Y 234.946,Z 411.221,A -85,B 0,C 180,E1 -19591.405,E2 -19591.405} C_VEL
LIN {X 0,Y 234.982,Z 411.214,A -85,B 0,C 180,E1 -19595.246,E2 -19595.246} C_VEL
LIN {X 0,Y 235.006,Z 411.213,A -85,B 0,C 180,E1 -19598.969,E2 -19598.969} C_VEL
LIN {X 0,Y 235.091,Z 411.202,A -85,B 0,C 180,E1 -19603.059,E2 -19603.059} C_VEL
LIN {X 0,Y 235.109,Z 411.197,A -85,B 0,C 180,E1 -19607.922,E2 -19607.922} C_VEL
LIN {X 0,Y 235.325,Z 411.169,A -85,B 0,C 180,E1 -19611.412,E2 -19611.412} C_VEL
LIN {X 0,Y 235.367,Z 411.16,A -85,B 0,C 180,E1 -19613.14,E2 -19613.14} C_VEL
LIN {X 0,Y 235.59,Z 411.138,A -85,B 0,C 180,E1 -19618.291,E2 -19618.291} C_VEL
LIN {X 0,Y 235.59,Z 411.133,A -85,B 0,C 180,E1 -19621.71,E2 -19621.71} C_VEL
LIN {X 0,Y 235.398,Z 411.163,A -85,B 0,C 180,E1 -19626.859,E2 -19626.859} C_VEL
LIN {X 0,Y 235.233,Z 411.183,A -85,B 0,C 180,E1 -19630.327,E2 -19630.327} C_VEL
LIN {X 0,Y 235.107,Z 411.195,A -85,B 0,C 180,E1 -19635.607,E2 -19635.607} C_VEL
LIN {X 0,Y 235.004,Z 411.209,A -85,B 0,C 180,E1 -19639.206,E2 -19639.206} C_VEL
LIN {X 0,Y 234.956,Z 411.209,A -85,B 0,C 180,E1 -19642.884,E2 -19642.884} C_VEL
LIN {X 0,Y 234.966,Z 411.217,A -85,B 0,C 180,E1 -19646.658,E2 -19646.658} C_VEL
LIN {X 0,Y 234.928,Z 411.216,A -85,B 0,C 180,E1 -19650.569,E2 -19650.569} C_VEL
LIN {X 0,Y 234.957,Z 411.216,A -85,B 0,C 180,E1 -19654.634,E2 -19654.634} C_VEL
LIN {X 0,Y 234.939,Z 411.216,A -85,B 0,C 180,E1 -19658.945,E2 -19658.945} C_VEL
LIN {X 0,Y 234.915,Z 411.22,A -85,B 0,C 180,E1 -19663.48,E2 -19663.48} C_VEL
LIN {X 0,Y 234.886,Z 411.225,A -85,B 0,C 180,E1 -19666.515,E2 -19666.515} C_VEL
LIN {X 0,Y 234.916,Z 411.205,A -85,B 0,C 180,E1 -19671.08,E2 -19671.08} C_VEL
LIN {X 0,Y 234.926,Z 411.214,A -85,B 0,C 180,E1 -19675.363,E2 -19675.363} C_VEL
LIN {X 0,Y 234.922,Z 411.224,A -85,B 0,C 180,E1 -19679.432,E2 -19679.432} C_VEL
LIN {X 0,Y 234.994,Z 411.201,A -85,B 0,C 180,E1 -19683.795,E2 -19683.795} C_VEL
LIN {X 0,Y 235.013,Z 411.21,A -85,B 0,C 180,E1 -19688.971,E2 -19688.971} C_VEL
LIN {X 0,Y 235.098,Z 411.19,A -85,B 0,C 180,E1 -19693.06,E2 -19693.06} C_VEL
LIN {X 0,Y 235.15,Z 411.191,A -85,B 0,C 180,E1 -19697.925,E2 -19697.925} C_VEL
LIN {X 0,Y 235.394,Z 411.164,A -85,B 0,C 180,E1 -19701.415,E2 -19701.415} C_VEL
LIN {X 0,Y 235.405,Z 411.162,A -85,B 0,C 180,E1 -19703.142,E2 -19703.142} C_VEL
LIN {X 0,Y 235.435,Z 411.158,A -85,B 0,C 180,E1 -19708.29,E2 -19708.29} C_VEL
LIN {X 0,Y 234.744,Z 411.379,A -85,B 0,C 180,E1 -19710,E2 -19710} C_VEL
LIN {X 0,Y 234.518,Z 413.033,A -85,B 0,C 180,E1 -19712.362,E2 -19712.362} C_VEL
LIN {X 0,Y 239.138,Z 426.622,A -85,B 0,C 180,E1 -19713.805,E2 -19713.805} C_VEL
LIN {X 0,Y 242.108,Z 438.124,A -85,B 0,C 180,E1 -19715.186,E2 -19715.186} C_VEL
LIN {X 0,Y 244.539,Z 449.592,A -85,B 0,C 180,E1 -19716.809,E2 -19716.809} C_VEL
LIN {X 0,Y 245.278,Z 454.751,A -85,B 0,C 180,E1 -19717.616,E2 -19717.616} C_VEL
LIN {X 0,Y 243.395,Z 466.066,A -85,B 0,C 180,E1 -19719.348,E2 -19719.348} C_VEL
LIN {X 0,Y 241.434,Z 476.211,A -85,B 0,C 180,E1 -19721.289,E2 -19721.289} C_VEL
LIN {X 0,Y 239.439,Z 485.755,A -85,B 0,C 180,E1 -19723.581,E2 -19723.581} C_VEL
LIN {X 0,Y 237.698,Z 493.411,A -85,B 0,C 180,E1 -19725.872,E2 -19725.872} C_VEL
LIN {X 0,Y 236.117,Z 500.351,A -85,B 0,C 180,E1 -19728.464,E2 -19728.464} C_VEL
LIN {X 0,Y 234.99,Z 505.774,A -85,B 0,C 180,E1 -19731.032,E2 -19731.032} C_VEL
LIN {X 0,Y 234.023,Z 510.457,A -85,B 0,C 180,E1 -19733.917,E2 -19733.917} C_VEL
LIN {X 0,Y 233.351,Z 513.831,A -85,B 0,C 180,E1 -19736.857,E2 -19736.857} C_VEL
LIN {X 0,Y 233.024,Z 515.512,A -85,B 0,C 180,E1 -19738.997,E2 -19738.997} C_VEL
LIN {X 0,Y 232.874,Z 516.892,A -85,B 0,C 180,E1 -19742.325,E2 -19742.325} C_VEL
LIN {X 0,Y 233.161,Z 516.819,A -85,B 0,C 180,E1 -19745.526,E2 -19745.526} C_VEL
LIN {X 0,Y 233.835,Z 515.482,A -85,B 0,C 180,E1 -19748.607,E2 -19748.607} C_VEL
LIN {X 0,Y 234.856,Z 512.971,A -85,B 0,C 180,E1 -19751.572,E2 -19751.572} C_VEL
LIN {X 0,Y 236.095,Z 509.346,A -85,B 0,C 180,E1 -19754.403,E2 -19754.403} C_VEL
LIN {X 0,Y 238.092,Z 503.641,A -85,B 0,C 180,E1 -19757.556,E2 -19757.556} C_VEL
LIN {X 0,Y 240.288,Z 497.222,A -85,B 0,C 180,E1 -19760.233,E2 -19760.233} C_VEL
LIN {X 0,Y 242.52,Z 490.295,A -85,B 0,C 180,E1 -19762.514,E2 -19762.514} C_VEL
LIN {X 0,Y 244.936,Z 482.059,A -85,B 0,C 180,E1 -19764.692,E2 -19764.692} C_VEL
LIN {X 0,Y 247.677,Z 471.869,A -85,B 0,C 180,E1 -19766.832,E2 -19766.832} C_VEL
LIN {X 0,Y 250.084,Z 461.488,A -85,B 0,C 180,E1 -19768.567,E2 -19768.567} C_VEL
LIN {X 0,Y 248.402,Z 450.935,A -85,B 0,C 180,E1 -19770.556,E2 -19770.556} C_VEL
LIN {X 0,Y 245.73,Z 440.66,A -85,B 0,C 180,E1 -19772.397,E2 -19772.397} C_VEL
LIN {X 0,Y 242.139,Z 430.659,A -85,B 0,C 180,E1 -19774.133,E2 -19774.133} C_VEL
LIN {X 0,Y 237.283,Z 420.359,A -85,B 0,C 180,E1 -19775.967,E2 -19775.967} C_VEL
LIN {X 0,Y 235.708,Z 417.487,A -85,B 0,C 180,E1 -19776.497,E2 -19776.497} C_VEL
LIN {X 0,Y 235.398,Z 416.272,A -85,B 0,C 180,E1 -19776.697,E2 -19776.697} C_VEL
LIN {X 0,Y 235.497,Z 415.161,A -85,B 0,C 180,E1 -19779.015,E2 -19779.015} C_VEL
LIN {X 0,Y 235.429,Z 413.491,A -85,B 0,C 180,E1 -19782.794,E2 -19782.794} C_VEL
LIN {X 0,Y 235.269,Z 412.178,A -85,B 0,C 180,E1 -19786.174,E2 -19786.174} C_VEL
LIN {X 0,Y 235.212,Z 411.187,A -85,B 0,C 180,E1 -19789.672,E2 -19789.672} C_VEL
LIN {X 0,Y 235.371,Z 411.165,A -85,B 0,C 180,E1 -19793.14,E2 -19793.14} C_VEL
LIN {X 0,Y 235.593,Z 411.139,A -85,B 0,C 180,E1 -19798.29,E2 -19798.29} C_VEL
LIN {X 0,Y 235.593,Z 411.136,A -85,B 0,C 180,E1 -19801.709,E2 -19801.709} C_VEL
LIN {X 0,Y 235.371,Z 411.166,A -85,B 0,C 180,E1 -19806.859,E2 -19806.859} C_VEL
LIN {X 0,Y 235.212,Z 411.181,A -85,B 0,C 180,E1 -19810.327,E2 -19810.327} C_VEL
LIN {X 0,Y 235.11,Z 411.194,A -85,B 0,C 180,E1 -19815.607,E2 -19815.607} C_VEL
LIN {X 0,Y 235.006,Z 411.206,A -85,B 0,C 180,E1 -19819.206,E2 -19819.206} C_VEL
LIN {X 0,Y 234.959,Z 411.219,A -85,B 0,C 180,E1 -19822.883,E2 -19822.883} C_VEL
LIN {X 0,Y 235.029,Z 411.504,A -85,B 0,C 180,E1 -19824.749,E2 -19824.749} C_VEL
LIN {X 0,Y 235.286,Z 413.193,A -85,B 0,C 180,E1 -19828.55,E2 -19828.55} C_VEL
LIN {X 0,Y 235.794,Z 415.876,A -85,B 0,C 180,E1 -19833.431,E2 -19833.431} C_VEL
LIN {X 0,Y 236.167,Z 417.889,A -85,B 0,C 180,E1 -19836.537,E2 -19836.537} C_VEL
LIN {X 0,Y 236.645,Z 421.028,A -85,B 0,C 180,E1 -19840.796,E2 -19840.796} C_VEL
LIN {X 0,Y 237.323,Z 424.801,A -85,B 0,C 180,E1 -19845.294,E2 -19845.294} C_VEL
LIN {X 0,Y 238.057,Z 428.712,A -85,B 0,C 180,E1 -19849.497,E2 -19849.497} C_VEL
LIN {X 0,Y 238.181,Z 430.42,A -85,B 0,C 180,E1 -19851.171,E2 -19851.171} C_VEL
LIN {X 0,Y 238.061,Z 431.694,A -85,B 0,C 180,E1 -19852.049,E2 -19852.049} C_VEL
LIN {X 0,Y 237.388,Z 434.618,A -85,B 0,C 180,E1 -19853.254,E2 -19853.254} C_VEL
LIN {X 0,Y 236.187,Z 439.849,A -85,B 0,C 180,E1 -19854.645,E2 -19854.645} C_VEL
LIN {X 0,Y 235.411,Z 446.15,A -85,B 0,C 180,E1 -19855.817,E2 -19855.817} C_VEL
LIN {X 0,Y 235.69,Z 451.302,A -85,B 0,C 180,E1 -19856.544,E2 -19856.544} C_VEL
LIN {X 0,Y 238.08,Z 463.343,A -85,B 0,C 180,E1 -19858.292,E2 -19858.292} C_VEL
LIN {X 0,Y 239.345,Z 474.789,A -85,B 0,C 180,E1 -19860.055,E2 -19860.055} C_VEL
LIN {X 0,Y 239.549,Z 484.36,A -85,B 0,C 180,E1 -19861.661,E2 -19861.661} C_VEL
LIN {X 0,Y 238.889,Z 494.718,A -85,B 0,C 180,E1 -19863.592,E2 -19863.592} C_VEL
LIN {X 0,Y 238.295,Z 499.93,A -85,B 0,C 180,E1 -19864.682,E2 -19864.682} C_VEL
LIN {X 0,Y 235.521,Z 509.082,A -85,B 0,C 180,E1 -19866.71,E2 -19866.71} C_VEL
LIN {X 0,Y 232.78,Z 518.006,A -85,B 0,C 180,E1 -19869.204,E2 -19869.204} C_VEL
LIN {X 0,Y 230.563,Z 525.352,A -85,B 0,C 180,E1 -19871.794,E2 -19871.794} C_VEL
LIN {X 0,Y 229.032,Z 530.323,A -85,B 0,C 180,E1 -19873.968,E2 -19873.968} C_VEL
LIN {X 0,Y 227.502,Z 535.198,A -85,B 0,C 180,E1 -19876.603,E2 -19876.603} C_VEL
LIN {X 0,Y 226.581,Z 538.987,A -85,B 0,C 180,E1 -19879.274,E2 -19879.274} C_VEL
LIN {X 0,Y 226.17,Z 540.973,A -85,B 0,C 180,E1 -19881.062,E2 -19881.062} C_VEL
LIN {X 0,Y 225.932,Z 542.528,A -85,B 0,C 180,E1 -19882.852,E2 -19882.852} C_VEL
LIN {X 0,Y 225.84,Z 543.711,A -85,B 0,C 180,E1 -19884.76,E2 -19884.76} C_VEL
LIN {X 0,Y 225.889,Z 544.731,A -85,B 0,C 180,E1 -19888.217,E2 -19888.217} C_VEL
LIN {X 0,Y 225.961,Z 544.664,A -85,B 0,C 180,E1 -19890,E2 -19890} C_VEL
LIN {X 0,Y 225.912,Z 544.147,A -85,B 0,C 180,E1 -19891.782,E2 -19891.782} C_VEL
LIN {X 0,Y 225.891,Z 543.229,A -85,B 0,C 180,E1 -19893.567,E2 -19893.567} C_VEL
LIN {X 0,Y 225.957,Z 541.74,A -85,B 0,C 180,E1 -19895.554,E2 -19895.554} C_VEL
LIN {X 0,Y 226.221,Z 537.869,A -85,B 0,C 180,E1 -19898.936,E2 -19898.936} C_VEL
LIN {X 0,Y 226.857,Z 533.599,A -85,B 0,C 180,E1 -19901.616,E2 -19901.616} C_VEL
LIN {X 0,Y 228.14,Z 527.117,A -85,B 0,C 180,E1 -19904.722,E2 -19904.722} C_VEL
LIN {X 0,Y 229.72,Z 520.001,A -85,B 0,C 180,E1 -19907.354,E2 -19907.354} C_VEL
LIN {X 0,Y 231.589,Z 511.616,A -85,B 0,C 180,E1 -19909.821,E2 -19909.821} C_VEL
LIN {X 0,Y 233.62,Z 502.019,A -85,B 0,C 180,E1 -19912.088,E2 -19912.088} C_VEL
LIN {X 0,Y 235.145,Z 494.366,A -85,B 0,C 180,E1 -19913.562,E2 -19913.562} C_VEL
LIN {X 0,Y 235.044,Z 484.032,A -85,B 0,C 180,E1 -19915.371,E2 -19915.371} C_VEL
LIN {X 0,Y 234.418,Z 472.605,A -85,B 0,C 180,E1 -19917.051,E2 -19917.051} C_VEL
LIN {X 0,Y 233,Z 460.366,A -85,B 0,C 180,E1 -19918.539,E2 -19918.539} C_VEL
LIN {X 0,Y 230.83,Z 447.185,A -85,B 0,C 180,E1 -19919.844,E2 -19919.844} C_VEL
LIN {X 0,Y 228.923,Z 437.657,A -85,B 0,C 180,E1 -19920.642,E2 -19920.642} C_VEL
LIN {X 0,Y 230.324,Z 431.844,A -85,B 0,C 180,E1 -19925.432,E2 -19925.432} C_VEL
LIN {X 0,Y 230.744,Z 429.245,A -85,B 0,C 180,E1 -19927.636,E2 -19927.636} C_VEL
LIN {X 0,Y 230.501,Z 426.255,A -85,B 0,C 180,E1 -19930.337,E2 -19930.337} C_VEL
LIN {X 0,Y 229.64,Z 421.652,A -85,B 0,C 180,E1 -19934.739,E2 -19934.739} C_VEL
LIN {X 0,Y 228.694,Z 416.719,A -85,B 0,C 180,E1 -19939.808,E2 -19939.808} C_VEL
LIN {X 0,Y 228.064,Z 412.781,A -85,B 0,C 180,E1 -19944.162,E2 -19944.162} C_VEL
LIN {X 0,Y 227.932,Z 412.094,A -85,B 0,C 180,E1 -19945.22,E2 -19945.22} C_VEL
LIN {X 0,Y 227.914,Z 412.097,A -85,B 0,C 180,E1 -19950.437,E2 -19950.437} C_VEL
LIN {X 0,Y 227.924,Z 412.095,A -85,B 0,C 180,E1 -19954.425,E2 -19954.425} C_VEL
LIN {X 0,Y 227.957,Z 412.089,A -85,B 0,C 180,E1 -19958.287,E2 -19958.287} C_VEL
LIN {X 0,Y 228.03,Z 412.082,A -85,B 0,C 180,E1 -19962.826,E2 -19962.826} C_VEL
LIN {X 0,Y 228.067,Z 412.074,A -85,B 0,C 180,E1 -19967.543,E2 -19967.543} C_VEL
LIN {X 0,Y 228.262,Z 412.05,A -85,B 0,C 180,E1 -19971.144,E2 -19971.144} C_VEL
LIN {X 0,Y 228.318,Z 412.039,A -85,B 0,C 180,E1 -19972.928,E2 -19972.928} C_VEL
LIN {X 0,Y 228.549,Z 412.015,A -85,B 0,C 180,E1 -19978.238,E2 -19978.238} C_VEL
LIN {X 0,Y 228.549,Z 412.01,A -85,B 0,C 180,E1 -19981.762,E2 -19981.762} C_VEL
LIN {X 0,Y 228.349,Z 412.04,A -85,B 0,C 180,E1 -19987.072,E2 -19987.072} C_VEL
LIN {X 0,Y 228.158,Z 412.061,A -85,B 0,C 180,E1 -19990.651,E2 -19990.651} C_VEL
LIN {X 0,Y 228.057,Z 412.069,A -85,B 0,C 180,E1 -19994.273,E2 -19994.273} C_VEL
LIN {X 0,Y 227.998,Z 412.084,A -85,B 0,C 180,E1 -19997.954,E2 -19997.954} C_VEL
LIN {X 0,Y 227.925,Z 412.085,A -85,B 0,C 180,E1 -20002.33,E2 -20002.33} C_VEL
LIN {X 0,Y 227.939,Z 412.092,A -85,B 0,C 180,E1 -20006.604,E2 -20006.604} C_VEL
LIN {X 0,Y 227.905,Z 412.093,A -85,B 0,C 180,E1 -20010.297,E2 -20010.297} C_VEL
LIN {X 0,Y 227.886,Z 412.091,A -85,B 0,C 180,E1 -20013.719,E2 -20013.719} C_VEL
LIN {X 0,Y 227.868,Z 412.102,A -85,B 0,C 180,E1 -20018.087,E2 -20018.087} C_VEL
LIN {X 0,Y 227.833,Z 412.102,A -85,B 0,C 180,E1 -20022.738,E2 -20022.738} C_VEL
LIN {X 0,Y 227.809,Z 412.105,A -85,B 0,C 180,E1 -20027.259,E2 -20027.259} C_VEL
LIN {X 0,Y 227.842,Z 412.082,A -85,B 0,C 180,E1 -20031.91,E2 -20031.91} C_VEL
LIN {X 0,Y 227.879,Z 412.099,A -85,B 0,C 180,E1 -20036.379,E2 -20036.379} C_VEL
LIN {X 0,Y 227.905,Z 412.096,A -85,B 0,C 180,E1 -20040.437,E2 -20040.437} C_VEL
LIN {X 0,Y 227.929,Z 412.079,A -85,B 0,C 180,E1 -20044.427,E2 -20044.427} C_VEL
LIN {X 0,Y 227.964,Z 412.09,A -85,B 0,C 180,E1 -20048.288,E2 -20048.288} C_VEL
LIN {X 0,Y 228.037,Z 412.069,A -85,B 0,C 180,E1 -20052.827,E2 -20052.827} C_VEL
LIN {X 0,Y 228.097,Z 412.073,A -85,B 0,C 180,E1 -20057.545,E2 -20057.545} C_VEL
LIN {X 0,Y 228.328,Z 412.043,A -85,B 0,C 180,E1 -20061.148,E2 -20061.148} C_VEL
LIN {X 0,Y 228.358,Z 412.039,A -85,B 0,C 180,E1 -20062.929,E2 -20062.929} C_VEL
LIN {X 0,Y 228.383,Z 412.037,A -85,B 0,C 180,E1 -20068.237,E2 -20068.237} C_VEL
LIN {X 0,Y 227.699,Z 412.39,A -85,B 0,C 180,E1 -20070,E2 -20070} C_VEL
